ELSIF (F_BACnet_GetObjType(_ObjectId) <> BACnetObjectType_Group) THEN
	(* wrong mapping / invalid object ID *)
	IF _ObjectId = 0 THEN
		nErrorId := BACnet_ERR_WRONG_MAPPING;
	ELSE
		nErrorId := BACnet_ERR_INVALID_OBJECTID;
	END_IF
	bReady := FALSE;
	tObjectID := 16#FFFFFFFF;

ELSE
	(* clear error flag *)
	nErrorId := BACnet_ERR_NO_ERROR;
	(* ready state *)
	bReady := TRUE;
	tObjectID := _ObjectId;
END_IF

(* set error flag *)
bError := (nErrorId <> BACnet_ERR_NO_ERROR);

END_FUNCTION_BLOCK

// POUs/BACnet Objects/Remote (Client)/Extended Process Data/FB_BACnet_RemoteLoop_EX
FUNCTION_BLOCK FB_BACnet_RemoteLoop_EX
VAR_IN_OUT
	RemoteDevice		: FB_BACnet_RemoteDevice;
END_VAR
VAR_OUTPUT
	bReady				: BOOL;
	fControlledValue	: REAL;
	fPresentValue		: REAL;
	bOverridden			: BOOL;
	bOutOfService		: BOOL;
	bFault				: BOOL;
	bInAlarm			: BOOL;
	bOpenLoop			: BOOL;
	bOtherFault			: BOOL;
	eEventState			: E_BACNETEVENTSTATE;
	tObjectID			: T_BACnet_ObjectIdentifier := 16#FFFFFFFF;
	bError				: BOOL;
	nErrorId			: UINT;
END_VAR
VAR
	_PresentValue AT%I*: REAL; 			(* ~(BACnet_PresentValue 				: LP	: )
			                               	(BACnet_RemoteCycletimeRead 		: 1000	: )
											(BACnet_RemoteFlagsRead        		: 1     : )
                                   			(BACnet_RemoteResubscriptionInterval: 240 	: )
		                                	(BACnet_RemoteCycleTimeWrite   		: 1000	: )
		                                	(BACnet_RemoteFlagsWrite       		: 1		: )	*)
	_ControlledVariableValue AT%I*: REAL;(* ~(BACnet_ControlledVariableValue 	:		: )	*)
	_ObjectId AT%I*: DWORD;				(* ~(BACnet_ObjectIdentifier			:		: LINK) *)
	_Reliability AT%I*: WORD;; 			(* ~(BACnet_Reliability 				:		: )	*)
	_StatusFlags AT%I*: WORD; 			(* ~(BACnet_StatusFlags 				:		: )	*)
	_EventState AT%I*: WORD;			(* ~(BACnet_EventState					:		: )	*)
	_nUpdateCount : UDINT := 0;
	_StatusFlagsBits : ST_BACnet_StatusFlags;
END_VAR

(* update client device *)
IF RemoteDevice._nUpdateCount = _nUpdateCount THEN
	RemoteDevice();
END_IF
(* remind current number of update counter *)
_nUpdateCount := RemoteDevice._nUpdateCount;

IF NOT RemoteDevice.bOperational THEN
	nErrorId := BACnet_ERR_OPERATIONAL;
	bReady := FALSE;

ELSIF (F_BACnet_GetObjType(_ObjectId) <> BACnetObjectType_Loop) THEN
	(* wrong mapping / invalid object ID *)
	IF _ObjectId = 0 THEN
		nErrorId := BACnet_ERR_WRONG_MAPPING;
	ELSE
		nErrorId := BACnet_ERR_INVALID_OBJECTID;
	END_IF
	bReady := FALSE;
	tObjectID := 16#FFFFFFFF;

ELSIF _StatusFlags >= 4 THEN
	(* clear error flag *)
	nErrorId := BACnet_ERR_NO_ERROR;
	(* ready state *)
	bReady := TRUE;

	(* present value *)
	fPresentValue := _PresentValue;
	fControlledValue := _ControlledVariableValue;

	(* build bit states *)
	_StatusFlagsBits := F_BACnet_StatusFlags(_StatusFlags);

	(* copy states to output *)
	bOverridden := _StatusFlagsBits.overridden;
	bOutOfService := _StatusFlagsBits.out_of_service;
	bFault := _StatusFlagsBits.fault;
	bInAlarm := _StatusFlagsBits.in_alarm;
	bOpenLoop := (_Reliability = TO_WORD(BACnetReliability_open_loop));
	bOtherFault := (_Reliability = TO_WORD(BACnetReliability_unreliable_other));
	eEventState := TO_INT(_EventState);
	tObjectID := _ObjectId;
ELSE
	(* server device not ready, reset local ready also *)
	bReady := FALSE;
	(* and set error ID *)
	nErrorId := BACnet_ERR_WRONG_MAPPING;
END_IF

(* set error flag *)
bError := (nErrorId <> BACnet_ERR_NO_ERROR);

END_FUNCTION_BLOCK

// POUs/BACnet Objects/Remote (Client)/Extended Process Data/FB_BACnet_RemoteMultiStateInput_EX
FUNCTION_BLOCK FB_BACnet_RemoteMultiStateInput_EX
VAR_IN_OUT
	RemoteDevice		: FB_BACnet_RemoteDevice;
END_VAR
VAR_OUTPUT
	bReady				: BOOL;
	nPresentValue		: UDINT;
	bOverridden			: BOOL;
	bOutOfService		: BOOL;
	bFault				: BOOL;
	bInAlarm			: BOOL;
	bOverRange			: BOOL;
	bUnderRange			: BOOL;
	bNoSensor			: BOOL;
	bOpenLoop			: BOOL;
	bShortedLoop		: BOOL;
	bMultiStateFault	: BOOL;
	bOtherFault			: BOOL;
	eEventState			: E_BACNETEVENTSTATE;
	nNbrOfStates		: UDINT;
	tObjectID			: T_BACnet_ObjectIdentifier := 16#FFFFFFFF;
	bError				: BOOL;
	nErrorId			: UINT;
END_VAR
VAR
	_PresentValue AT%I*: UDINT; 		(* ~(BACnet_PresentValue 				:		: )
								   			(BACnet_ObjectType 					: MI	: )
											(BACnet_RemoteCycletimeRead 		: 1000	: )
											(BACnet_RemoteFlagsRead        		: 1		: )
											(BACnet_RemoteResubscriptionInterval: 240	: )
                                			(BACnet_RemoteCycleTimeWrite   		: 1000	: )
                                			(BACnet_RemoteFlagsWrite       		: 1		: )	*)
	_NumberOfStates AT%I*: UDINT;		(* ~(BACnet_NumberOfStates				:		: )	*)
	_ObjectId AT%I*: DWORD;				(* ~(BACnet_ObjectIdentifier			:		: LINK) *)
	_StatusFlags AT%I*: WORD; 			(* ~(BACnet_StatusFlags 				:		: )	*)
	_Reliability AT%I*: WORD;; 			(* ~(BACnet_Reliability 				:		: )	*)
	_EventState AT%I*: WORD; 			(* ~(BACnet_EventState 					:		: )	*)
	_nUpdateCount : UDINT := 0;
	_StatusFlagsBits : ST_BACnet_StatusFlags;
END_VAR

(* update client device *)
IF RemoteDevice._nUpdateCount = _nUpdateCount THEN
	RemoteDevice();
END_IF
(* remind current number of update counter *)
_nUpdateCount := RemoteDevice._nUpdateCount;

IF NOT RemoteDevice.bOperational THEN
	nErrorId := BACnet_ERR_OPERATIONAL;
	bReady := FALSE;

ELSIF (F_BACnet_GetObjType(_ObjectId) <> BACnetObjectType_MultiStateInput) THEN
	(* wrong mapping / invalid object ID *)
	IF _ObjectId = 0 THEN
		nErrorId := BACnet_ERR_WRONG_MAPPING;
	ELSE
		nErrorId := BACnet_ERR_INVALID_OBJECTID;
	END_IF
	bReady := FALSE;
	tObjectID := 16#FFFFFFFF;

ELSIF _StatusFlags >= 4 THEN
	(* clear error flag *)
	nErrorId := BACnet_ERR_NO_ERROR;
	(* ready state *)
	bReady := TRUE;

	(* present value *)
	nPresentValue := _PresentValue;

	(* build bit states *)
	_StatusFlagsBits := F_BACnet_StatusFlags(_StatusFlags);

	(* copy states to output *)
	bOverridden := _StatusFlagsBits.overridden;
	bOutOfService := _StatusFlagsBits.out_of_service;
	bFault := _StatusFlagsBits.fault;
	bInAlarm := _StatusFlagsBits.in_alarm;
	bOverRange := (_Reliability = TO_WORD(BACnetReliability_over_range));
	bUnderRange := (_Reliability = TO_WORD(BACnetReliability_under_range));
	bNoSensor := (_Reliability = TO_WORD(BACnetReliability_no_sensor));
	bOpenLoop := (_Reliability = TO_WORD(BACnetReliability_open_loop));
	bShortedLoop := (_Reliability = TO_WORD(BACnetReliability_shorted_loop));
	bMultiStateFault := (_Reliability = TO_WORD(BACnetReliability_multi_state_fault));
	bOtherFault := (_Reliability = TO_WORD(BACnetReliability_unreliable_other));
	nNbrOfStates := _NumberOfStates;
	eEventState := TO_INT(_EventState);
	tObjectID := _ObjectId;

ELSE
	(* server device not ready, reset local ready also *)
	bReady := FALSE;
	(* and set error ID *)
	nErrorId := BACnet_ERR_WRONG_MAPPING;
END_IF

(* set error flag *)
bError := (nErrorId <> BACnet_ERR_NO_ERROR);

END_FUNCTION_BLOCK

// POUs/BACnet Objects/Remote (Client)/Extended Process Data/FB_BACnet_RemoteMultiStateOutput_EX
FUNCTION_BLOCK FB_BACnet_RemoteMultiStateOutput_EX
VAR_INPUT
	bEnablePV			: BOOL; (* enable present value with priority x in priority array, FALSE = priority x disable *)
	bNullPV				: BOOL; (* clear priority entry *)
	nPV					: UDINT; (* number for priority x, when input bEnablePV is TRUE *)
END_VAR
VAR_IN_OUT
	RemoteDevice		: FB_BACnet_RemoteDevice;
END_VAR
VAR_OUTPUT
	bReady				: BOOL;
	nPresentValue		: UDINT;
	bOverridden			: BOOL;
	bOutOfService		: BOOL;
	bFault				: BOOL;
	bInAlarm			: BOOL;
	bNoOutput			: BOOL;
	bOpenLoop			: BOOL;
	bShortedLoop		: BOOL;
	bOtherFault			: BOOL;
	eEventState			: E_BACNETEVENTSTATE;
	nActivePrio			: UINT;
	nNbrOfStates		: UDINT;
	tObjectID			: T_BACnet_ObjectIdentifier := 16#FFFFFFFF;
	bError				: BOOL;
	nErrorId			: UINT;
END_VAR
VAR
	_PresentValue AT%I*: UDINT; 		(* ~(BACnet_PresentValue 				:		: )
								   			(BACnet_ObjectType					: MO	: )
											(BACnet_RemoteCycletimeRead 		: 1000	: )
											(BACnet_RemoteFlagsRead        		: 1		: )
											(BACnet_RemoteResubscriptionInterval: 240	: )
		                                	(BACnet_RemoteCycleTimeWrite   		: 1000	: )
		                                	(BACnet_RemoteFlagsWrite       		: 1		: )	*)
	_NumberOfStates AT%I*: UDINT;		(* ~(BACnet_NumberOfStates				:		: )	*)
	_ActivePriority AT%I*: UDINT; 		(* ~(BACnet_ActivePriority 				:		: )	*)
	_ObjectId AT%I*: DWORD;				(* ~(BACnet_ObjectIdentifier			:		: LINK) *)
	_StatusFlags AT%I*: WORD; 			(* ~(BACnet_StatusFlags					:		: )	*)
	_Reliability AT%I*: WORD;; 			(* ~(BACnet_Reliability					:		: )	*)
	_EventState AT%I*: WORD;			(* ~(BACnet_EventState					:		: )	*)
    _PresentValue_Priority12 AT%Q*: UDINT;(* ~(BACnet_PresentValue_Priority12	:		: )	*)
	_nUpdateCount : UDINT := 0;
	_StatusFlagsBits : ST_BACnet_StatusFlags;
END_VAR

(* update client device *)
IF RemoteDevice._nUpdateCount = _nUpdateCount THEN
	RemoteDevice();
END_IF
(* remind current number of update counter *)
_nUpdateCount := RemoteDevice._nUpdateCount;

IF RemoteDevice.bFirstCycle THEN
	(* first call of the server device since reboot/reset *)
	bReady := FALSE;
	_PresentValue_Priority12 := 16#FFFFFFFF;
ELSIF NOT RemoteDevice.bOperational THEN
	nErrorId := BACnet_ERR_OPERATIONAL;
	bReady := FALSE;

ELSIF (F_BACnet_GetObjType(_ObjectId) <> BACnetObjectType_MultiStateOutput) THEN
	(* wrong mapping / invalid object ID *)
	IF _ObjectId = 0 THEN
		nErrorId := BACnet_ERR_WRONG_MAPPING;
	ELSE
		nErrorId := BACnet_ERR_INVALID_OBJECTID;
	END_IF
	bReady := FALSE;
	tObjectID := 16#FFFFFFFF;

ELSIF _StatusFlags >= 4 THEN
	(* clear error flag *)
	nErrorId := BACnet_ERR_NO_ERROR;
	(* ready state *)
	bReady := TRUE;

	(* write into priority array *)
	_PresentValue_Priority12 := F_BACnet_MultiStatePV(bEnablePV, bNullPV, nPV);

	(* present value *)
	nPresentValue := _PresentValue;

	(* build bit states *)
	_StatusFlagsBits := F_BACnet_StatusFlags(_StatusFlags);

	(* copy states to output *)
	bOverridden := _StatusFlagsBits.overridden;
	bOutOfService := _StatusFlagsBits.out_of_service;
	bFault := _StatusFlagsBits.fault;
	bInAlarm := _StatusFlagsBits.in_alarm;
	bNoOutput := (_Reliability = TO_WORD(BACnetReliability_no_output));
	bOpenLoop := (_Reliability = TO_WORD(BACnetReliability_open_loop));
	bShortedLoop := (_Reliability = TO_WORD(BACnetReliability_shorted_loop));
	bOtherFault := (_Reliability = TO_WORD(BACnetReliability_unreliable_other));
	eEventState := TO_INT(_EventState);
	tObjectID := _ObjectId;

	(* copy active priority *)
	nActivePrio := UDINT_TO_UINT(_ActivePriority);

	(* number of states *)
	nNbrOfStates := _NumberOfStates;

ELSE
	(* server device not ready, reset local ready also *)
	bReady := FALSE;
	(* and set error ID *)
	nErrorId := BACnet_ERR_WRONG_MAPPING;
END_IF

(* set error flag *)
bError := (nErrorId <> BACnet_ERR_NO_ERROR);

END_FUNCTION_BLOCK

// POUs/BACnet Objects/Remote (Client)/Extended Process Data/FB_BACnet_RemoteMultiStateValue_EX
FUNCTION_BLOCK FB_BACnet_RemoteMultiStateValue_EX
VAR_INPUT
	bEnablePV			: BOOL; (* enable present value with priority x in priority array, FALSE = priority x disable *)
	bNullPV				: BOOL; (* clear priority entry *)
	nPV					: UDINT; (* number for priority x, when input bEnablePV is TRUE *)
END_VAR
VAR_IN_OUT
	RemoteDevice		: FB_BACnet_RemoteDevice;
END_VAR
VAR_OUTPUT
	bReady				: BOOL;
	nPresentValue		: UDINT;
	bOverridden			: BOOL;
	bOutOfService		: BOOL;
	bFault				: BOOL;
	bInAlarm			: BOOL;
	bMultiStateFault	: BOOL;
	bOtherFault			: BOOL;
	eEventState			: E_BACNETEVENTSTATE;
	nNbrOfStates		: UDINT;
	tObjectID			: T_BACnet_ObjectIdentifier := 16#FFFFFFFF;
	bError				: BOOL;
	nErrorId			: UINT;
END_VAR
VAR
	_PresentValue AT%I*: UDINT; 		(* ~(BACnet_PresentValue 				:		: )
											(BACnet_ObjectType 					: MV	: )
											(BACnet_RemoteCycletimeRead 		: 1000	: )
											(BACnet_RemoteFlagsRead        		: 1		: )
											(BACnet_RemoteResubscriptionInterval: 240	: )
											(BACnet_RemoteCycleTimeWrite   		: 1000	: )
											(BACnet_RemoteFlagsWrite       		: 1		: )	*)
	_NumberOfStates AT%I*: UDINT;		(* ~(BACnet_NumberOfStates				:		: )	*)
	_EventState AT%I*: WORD;			(* ~(BACnet_EventState					:		: )	*)
	_ObjectId AT%I*: DWORD;				(* ~(BACnet_ObjectIdentifier			:		: LINK) *)
	_StatusFlags AT%I*: WORD;			(* ~(BACnet_StatusFlags 				:		: )	*)
	_Reliability AT%I*: WORD;;			(* ~(BACnet_Reliability 				:		: )	*)
    _PresentValue_Priority12 AT%Q*: UDINT;(* ~(BACnet_PresentValue_Priority12	:		: )	*)
	_nUpdateCount : UDINT := 0;
	_StatusFlagsBits : ST_BACnet_StatusFlags;
END_VAR

(* update client device *)
IF RemoteDevice._nUpdateCount = _nUpdateCount THEN
	RemoteDevice();
END_IF
(* remind current number of update counter *)
_nUpdateCount := RemoteDevice._nUpdateCount;

IF RemoteDevice.bFirstCycle THEN
	(* first call of the server device since reboot/reset *)
	bReady := FALSE;
	_PresentValue_Priority12 := 16#FFFFFFFF;
ELSIF NOT RemoteDevice.bOperational THEN
	nErrorId := BACnet_ERR_OPERATIONAL;
	bReady := FALSE;

ELSIF (F_BACnet_GetObjType(_ObjectId) <> BACnetObjectType_MultiStateValue) THEN
	(* wrong mapping / invalid object ID *)
	IF _ObjectId = 0 THEN
		nErrorId := BACnet_ERR_WRONG_MAPPING;
	ELSE
		nErrorId := BACnet_ERR_INVALID_OBJECTID;
	END_IF
	bReady := FALSE;
	tObjectID := 16#FFFFFFFF;

ELSIF _StatusFlags >= 4 THEN
	(* clear error flag *)
	nErrorId := BACnet_ERR_NO_ERROR;
	(* ready state *)
	bReady := TRUE;

	(* write into priority array *)
	_PresentValue_Priority12 := F_BACnet_MultiStatePV(bEnablePV, bNullPV, nPV);

	(* present value *)
	nPresentValue := _PresentValue;

	(* build bit states *)
	_StatusFlagsBits := F_BACnet_StatusFlags(_StatusFlags);

	(* copy states to output *)
	bOverridden := _StatusFlagsBits.overridden;
	bOutOfService := _StatusFlagsBits.out_of_service;
	bFault := _StatusFlagsBits.fault;
	bInAlarm := _StatusFlagsBits.in_alarm;
	bMultiStateFault := (_Reliability = TO_WORD(BACnetReliability_multi_state_fault));
	bOtherFault := (_Reliability = TO_WORD(BACnetReliability_unreliable_other));
	eEventState := TO_INT(_EventState);
	tObjectID := _ObjectId;

	(* number of states *)
	nNbrOfStates := _NumberOfStates;

ELSE
	(* server device not ready, reset local ready also *)
	bReady := FALSE;
	(* and set error ID *)
	nErrorId := BACnet_ERR_WRONG_MAPPING;
END_IF

(* set error flag *)
bError := (nErrorId <> BACnet_ERR_NO_ERROR);

END_FUNCTION_BLOCK

// POUs/BACnet Objects/Remote (Client)/Extended Process Data/FB_BACnet_RemoteNotificationClass_EX
FUNCTION_BLOCK FB_BACnet_RemoteNotificationClass_EX
VAR_IN_OUT
	RemoteDevice		: FB_BACnet_RemoteDevice;
END_VAR
VAR_OUTPUT
	bReady				: BOOL;
	tObjectID			: T_BACnet_ObjectIdentifier := 16#FFFFFFFF;
	bError				: BOOL;
	nErrorId			: UINT;
END_VAR
VAR
	_ObjectId AT%I*: DWORD;				(* ~(BACnet_ObjectIdentifier	:		: LINK)
											(BACNET_OBJECTTYPE			: NC	: ) *)
	_nUpdateCount : UDINT := 0;
END_VAR

(* update client device *)
IF RemoteDevice._nUpdateCount = _nUpdateCount THEN
	RemoteDevice();
END_IF
(* remind current number of update counter *)
_nUpdateCount := RemoteDevice._nUpdateCount;

IF NOT RemoteDevice.bOperational THEN
	(* server device not ready, reset local ready also *)
	bReady := FALSE;
	(* and set error ID *)
	nErrorId := BACnet_ERR_OPERATIONAL;

ELSIF (F_BACnet_GetObjType(_ObjectId) <> BACnetObjectType_NotificationClass) THEN
	(* wrong mapping / invalid object ID *)
	IF _ObjectId = 0 THEN
		nErrorId := BACnet_ERR_WRONG_MAPPING;
	ELSE
		nErrorId := BACnet_ERR_INVALID_OBJECTID;
	END_IF
	bReady := FALSE;
	tObjectID := 16#FFFFFFFF;

ELSIF RemoteDevice.bOperational THEN
	(* clear error flag *)
	nErrorId := BACnet_ERR_NO_ERROR;
	(* ready state *)
	bReady := TRUE;
	tObjectID := _ObjectId;

END_IF

(* set error flag *)
bError := (nErrorId <> BACnet_ERR_NO_ERROR);

END_FUNCTION_BLOCK

// POUs/BACnet Objects/Remote (Client)/Extended Process Data/FB_BACnet_RemoteProgram_EX
FUNCTION_BLOCK FB_BACnet_RemoteProgram_EX
VAR_INPUT
	bEnablePV			: BOOL;
	ePV					: E_BACNETPROGRAMREQUEST;
	bRetrigger			: BOOL; (* execute selected request on raising edge again *)
END_VAR
VAR_IN_OUT
	RemoteDevice		: FB_BACnet_RemoteDevice;
END_VAR
VAR_OUTPUT
	bReady				: BOOL;
	ePrgState			: E_BACNETPROGRAMSTATE;
	ePrgChangeReq		: E_BACNETPROGRAMREQUEST;
	ePrgReasonHalt		: E_BACNETPROGRAMERROR;
	bOverridden			: BOOL;
	bOutOfService		: BOOL;
	bFault				: BOOL;
	bInAlarm			: BOOL;
	bProcessError		: BOOL;
	bOtherFault			: BOOL;
	tObjectID		: T_BACnet_ObjectIdentifier := 16#FFFFFFFF;
	bError				: BOOL;
	nErrorId			: UINT;
END_VAR
VAR
	_ProgramState AT%I*: WORD;			(* ~(BACnet_ProgramState 				:		: )
											(BACnet_ObjectType 					: PROG	: )
											(BACnet_RemoteCycletimeRead 		: 1000	: )
											(BACnet_RemoteFlagsRead        		: 1    	: )
											(BACnet_RemoteResubscriptionInterval: 240 	: )
											(BACnet_RemoteCycleTimeWrite   		: 1000	: )
											(BACnet_RemoteFlagsWrite       		: 1		: )	*)
	_ProgramChangeState AT%I*: WORD;	(* ~(BACnet_ProgramChange 				:		: )	*)
	_ReasonForHalt AT%I*: WORD;			(* ~(BACnet_ReasonForHalt 				: 		: )	*)
	_StatusFlags AT%I*: WORD;			(* ~(BACnet_StatusFlags 				:		: )	*)
	_Reliability AT%I*: WORD;;			(* ~(BACnet_Reliability 				:		: )	*)
	_ProgramChangeRequest AT%Q*: WORD;	(* ~(BACnet_ProgramChange 				:		: )	*)
	_ObjectId AT%I*: DWORD;				(* ~(BACnet_ObjectIdentifier			:		: LINK) *)
	_nUpdateCount : UDINT := 0;
	_StatusFlagsBits : ST_BACnet_StatusFlags;
	_rtrigRetriggerPv : R_TRIG;
END_VAR

(* update client device *)
IF RemoteDevice._nUpdateCount = _nUpdateCount THEN
	RemoteDevice();
END_IF
(* remind current number of update counter *)
_nUpdateCount := RemoteDevice._nUpdateCount;

(* call trigger *)
_rtrigRetriggerPv(CLK:= bRetrigger, Q=> );

IF RemoteDevice.bFirstCycle THEN
	(* first call of the server device since reboot/reset *)
	bReady := FALSE;
	_ProgramChangeRequest := 0;
ELSIF NOT RemoteDevice.bOperational THEN
	nErrorId := BACnet_ERR_OPERATIONAL;
	bReady := FALSE;

ELSIF (F_BACnet_GetObjType(_ObjectId) <> BACnetObjectType_Program) THEN
	(* wrong mapping / invalid object ID *)
	IF _ObjectId = 0 THEN
		nErrorId := BACnet_ERR_WRONG_MAPPING;
	ELSE
		nErrorId := BACnet_ERR_INVALID_OBJECTID;
	END_IF
	bReady := FALSE;
	tObjectID := 16#FFFFFFFF;

ELSIF _StatusFlags >= 4 THEN
	(* clear error flag *)
	nErrorId := BACnet_ERR_NO_ERROR;

	(* ready state *)
	bReady := TRUE;

	(* decode status flags *)
	_StatusFlagsBits := F_BACnet_StatusFlags(_StatusFlags);

	(* copy states to output *)
	bOverridden := _StatusFlagsBits.overridden;
	bOutOfService := _StatusFlagsBits.out_of_service;
	bFault := _StatusFlagsBits.fault;
	bInAlarm := _StatusFlagsBits.in_alarm;
	bProcessError := (_Reliability = TO_WORD(BACnetReliability_process_error));
	bOtherFault := (_Reliability = TO_WORD(BACnetReliability_unreliable_other));
	tObjectID := _ObjectId;

	(* present value from BACnet *)
	ePrgState := TO_INT(_ProgramState);
	(* present value to BACnet *)
	IF bEnablePV THEN
		IF _rtrigRetriggerPv.Q THEN
			(* trigger request *)
			_ProgramChangeRequest := 0;
		ELSE
			(* set request value *)
			_ProgramChangeRequest := TO_WORD(ePV);
		END_IF
	ELSE
		_ProgramChangeRequest := 0;
	END_IF
	(* other states *)
	ePrgReasonHalt := TO_INT(_ReasonForHalt);
	ePrgChangeReq := TO_INT(_ProgramChangeState);

ELSE
	(* server device not ready, reset local ready also *)
	bReady := FALSE;
	(* and set error ID *)
	nErrorId := BACnet_ERR_WRONG_MAPPING;
END_IF

(* set error flag *)
bError := (nErrorId <> BACnet_ERR_NO_ERROR);

END_FUNCTION_BLOCK

// POUs/BACnet Objects/Remote (Client)/Extended Process Data/FB_BACnet_RemotePulseConverter_EX
FUNCTION_BLOCK FB_BACnet_RemotePulseConverter_EX
VAR_IN_OUT
	RemoteDevice	: FB_BACnet_RemoteDevice;
END_VAR
VAR_OUTPUT
	bReady			: BOOL;
	fPresentValue	: REAL;
	nCount			: UDINT;
	bOverridden		: BOOL;
	bOutOfService	: BOOL;
	bFault			: BOOL;
	bInAlarm		: BOOL;
	bOverRange		: BOOL;
	bUnderRange		: BOOL;
	bNoSensor		: BOOL;
	bOpenLoop		: BOOL;
	bShortedLoop	: BOOL;
	bCommFailure	: BOOL;
	bConfigError	: BOOL;
	bOtherFault		: BOOL;
	tObjectID		: T_BACnet_ObjectIdentifier := 16#FFFFFFFF;
	bError			: BOOL;
	nErrorId		: UINT;
END_VAR
VAR
	_ObjectId AT%I*: DWORD;		(* ~(BACnet_ObjectIdentifier			:		: LINK) *)
	_Count AT%I*: UDINT;		(* ~(BACnet_Count		 				:		: ) *)
	_PresentValue AT%I*: REAL;	(* ~(BACnet_PresentValue 				:		: )	*)
	_StatusFlags AT%I*: UINT;	(* ~(BACnet_StatusFlags 				:		: )
									(BACnet_ObjectType 					: PC	: )
									(BACnet_RemoteCycletimeRead 		: 1000	: )
									(BACnet_RemoteFlagsRead        		: 1		: )
									(BACnet_RemoteResubscriptionInterval: 240	: )
                                	(BACnet_RemoteCycleTimeWrite   		: 1000	: )
                                	(BACnet_RemoteFlagsWrite       		: 1		: )	*)
	_Reliability AT%I*:WORD;	(* ~(BACnet_Reliability					:		: )	*)
	_StatusFlagsBits : ST_BACnet_StatusFlags;
	_nUpdateCount : UDINT := 0;
END_VAR

(* update client device *)
IF RemoteDevice._nUpdateCount = _nUpdateCount THEN
	RemoteDevice();
END_IF
(* remind current number of update counter *)
_nUpdateCount := RemoteDevice._nUpdateCount;

IF NOT RemoteDevice.bOperational THEN
	nErrorId := BACnet_ERR_OPERATIONAL;
	bReady := FALSE;

ELSIF (F_BACnet_GetObjType(_ObjectId) <> BACnetObjectType_PulseConverter) THEN
	(* wrong mapping / invalid object ID *)
	IF _ObjectId = 0 THEN
		nErrorId := BACnet_ERR_WRONG_MAPPING;
	ELSE
		nErrorId := BACnet_ERR_INVALID_OBJECTID;
	END_IF
	bReady := FALSE;
	tObjectID := 16#FFFFFFFF;

ELSIF _StatusFlags >= 4 THEN
	(* clear error flag *)
	nErrorId := BACnet_ERR_NO_ERROR;
	(* ready state *)
	bReady := TRUE;

	(* present value *)
	fPresentValue := _PresentValue;
	nCount := _Count;

	(* build bit states *)
	_StatusFlagsBits := F_BACnet_StatusFlags(_StatusFlags);

	(* copy states to output *)
	bOverridden := _StatusFlagsBits.overridden;
	bOutOfService := _StatusFlagsBits.out_of_service;
	bFault := _StatusFlagsBits.fault;
	bInAlarm := _StatusFlagsBits.in_alarm;
	tObjectID := _ObjectId;

	(* reliability *)
	bOverRange	:= (_Reliability = TO_WORD(BACnetReliability_over_range));
	bUnderRange	:= (_Reliability = TO_WORD(BACnetReliability_under_range));
	bNoSensor	:= (_Reliability = TO_WORD(BACnetReliability_no_sensor));
	bOpenLoop	:= (_Reliability = TO_WORD(BACnetReliability_open_loop));
	bShortedLoop:= (_Reliability = TO_WORD(BACnetReliability_shorted_loop));
	bCommFailure := (_Reliability = TO_WORD(BACnetReliability_communication_failure));
	bConfigError:= (_Reliability = TO_WORD(BACnetReliability_configuration_error));
	bOtherFault	:= (_Reliability = TO_WORD(BACnetReliability_unreliable_other));

ELSE
	(* server device not ready, reset local ready also *)
	bReady := FALSE;
	(* and set error ID *)
	nErrorId := BACnet_ERR_WRONG_MAPPING;
END_IF

(* set error flag *)
bError := (nErrorId <> BACnet_ERR_NO_ERROR);

END_FUNCTION_BLOCK

// POUs/BACnet Objects/Remote (Client)/Extended Process Data/FB_BACnet_RemoteSchedule_EX
FUNCTION_BLOCK FB_BACnet_RemoteSchedule_EX
VAR_IN_OUT
	RemoteDevice			: FB_BACnet_RemoteDevice;
END_VAR
VAR_OUTPUT
	bReady				: BOOL;
	bPresentValue		: BOOL;
	bOverridden			: BOOL;
	bOutOfService		: BOOL;
	bFault				: BOOL;
	bInAlarm			: BOOL;
	bConfigError		: BOOL;
	bOtherFault			: BOOL;
	tObjectID			: T_BACnet_ObjectIdentifier := 16#FFFFFFFF;
	bError				: BOOL;
	nErrorId			: UINT;
END_VAR
VAR
	_ObjectId AT%I*: DWORD;				(* ~(BACnet_ObjectIdentifier			:		: LINK) *)
	_Reliability AT%I*: WORD;; 			(* ~(BACnet_Reliability 				:		: )	*)
	_StatusFlags AT%I*: WORD; 			(* ~(BACnet_StatusFlags 				:		: )	*)
	_PresentValue AT%I*: BOOL;			(* ~(BACnet_PresentValueBool 			:		: )
											(BACnet_ObjectType 					: SCHED	: )
											(BACnet_RemoteCycletimeRead 		: 1000	: )
											(BACnet_RemoteFlagsRead        		: 1		: )
											(BACnet_RemoteResubscriptionInterval: 240	: )
                            				(BACnet_RemoteCycleTimeWrite   		: 1000	: )
                            				(BACnet_RemoteFlagsWrite       		: 1		: )	*)
	_StatusFlagsBits : ST_BACnet_StatusFlags;
	_nUpdateCount : UDINT := 0;
END_VAR

(* update client device *)
IF RemoteDevice._nUpdateCount = _nUpdateCount THEN
	RemoteDevice();
END_IF
(* remind current number of update counter *)
_nUpdateCount := RemoteDevice._nUpdateCount;

IF NOT RemoteDevice.bOperational THEN
	nErrorId := BACnet_ERR_OPERATIONAL;
	bReady := FALSE;

ELSIF (F_BACnet_GetObjType(_ObjectId) <> BACnetObjectType_Schedule) THEN
	(* wrong mapping / invalid object ID *)
	IF _ObjectId = 0 THEN
		nErrorId := BACnet_ERR_WRONG_MAPPING;
	ELSE
		nErrorId := BACnet_ERR_INVALID_OBJECTID;
	END_IF
	bReady := FALSE;
	tObjectID := 16#FFFFFFFF;

ELSIF _StatusFlags >= 4 THEN
	(* clear error flag *)
	nErrorId := BACnet_ERR_NO_ERROR;
	(* ready state *)
	bReady := TRUE;

	(* present value *)
	bPresentValue := _PresentValue;

	(* build bit states *)
	_StatusFlagsBits := F_BACnet_StatusFlags(_StatusFlags);

	(* copy states to output *)
	bOverridden := _StatusFlagsBits.overridden;
	bOutOfService := _StatusFlagsBits.out_of_service;
	bFault := _StatusFlagsBits.fault;
	bInAlarm := _StatusFlagsBits.in_alarm;
	bConfigError := (_Reliability = TO_WORD(BACnetReliability_configuration_error));
	bOtherFault := (_Reliability = TO_WORD(BACnetReliability_unreliable_other));
	tObjectID := _ObjectId;

ELSE
	bReady := FALSE;
	(* and set error ID *)
	nErrorId := BACnet_ERR_WRONG_MAPPING;
END_IF

(* set error flag *)
bError := (nErrorId <> BACnet_ERR_NO_ERROR);

END_FUNCTION_BLOCK

// POUs/BACnet Objects/Remote (Client)/Extended Process Data/FB_BACnet_RemoteTrendLog_EX
FUNCTION_BLOCK FB_BACnet_RemoteTrendLog_EX
VAR_OUTPUT
	bReady				: BOOL;
	bLogEnable			: BOOL;
	nRecordCount		: UDINT;
	nTotalCount			: UDINT;
	eEventState			: E_BACNETEVENTSTATE;
	tObjectID			: T_BACnet_ObjectIdentifier := 16#FFFFFFFF;
	bError				: BOOL;
	nErrorId			: UINT;
END_VAR
VAR_IN_OUT
	RemoteDevice			: FB_BACnet_RemoteDevice;
END_VAR
VAR
	_RecordCount AT%I*: UDINT;			(* ~(BACnet_RecordCount					:		: )
											(BACnet_ObjectType					: TLOG	: )
											(BACnet_RemoteCycletimeRead 		: 1000	: )
											(BACnet_RemoteFlagsRead        		: 1		: )
											(BACnet_RemoteResubscriptionInterval: 240	: )
											(BACnet_RemoteCycleTimeWrite   		: 1000	: )
                                			(BACnet_RemoteFlagsWrite       		: 1		: )	*)
	_TotalRecordCount AT%I*: UDINT;		(* ~(BACnet_TotalRecordCount			:		: )	*)
	_ObjectId AT%I*: DWORD;				(* ~(BACnet_ObjectIdentifier			:		: LINK) *)
	_EventState AT%I*: WORD;			(* ~(BACnet_EventState					:		: )	*)
	_LogEnable AT%I*: BOOL;				(* ~(BACnet_LogEnable					: 		: )	*)
	_nUpdateCount : UDINT := 0;
END_VAR

(* update client device *)
IF RemoteDevice._nUpdateCount = _nUpdateCount THEN
	RemoteDevice();
END_IF
(* remind current number of update counter *)
_nUpdateCount := RemoteDevice._nUpdateCount;

IF NOT RemoteDevice.bOperational THEN
	(* mapping seems to be wrong *)
	nErrorId := BACnet_ERR_OPERATIONAL;
	bReady := FALSE;

ELSIF (F_BACnet_GetObjType(_ObjectId) <> BACnetObjectType_TrendLog) THEN
	(* wrong mapping / invalid object ID *)
	IF _ObjectId = 0 THEN
		nErrorId := BACnet_ERR_WRONG_MAPPING;
	ELSE
		nErrorId := BACnet_ERR_INVALID_OBJECTID;
	END_IF
	bReady := FALSE;
	tObjectID := 16#FFFFFFFF;

ELSIF _EventState >= 0 THEN
	(* clear error flag *)
	nErrorId := BACnet_ERR_NO_ERROR;
	(* ready state *)
	bReady := TRUE;

	(* convert enumeration *)
	eEventState := TO_INT(_EventState);

	(* other states *)
	nRecordCount := _RecordCount;
	nTotalCount := _TotalRecordCount;
	bLogEnable := _LogEnable;
	tObjectID := _ObjectId;

ELSE
	bReady := FALSE;
	(* and set error ID *)
	nErrorId := BACnet_ERR_WRONG_MAPPING;
END_IF

(* set error flag *)
bError := (nErrorId <> BACnet_ERR_NO_ERROR);

END_FUNCTION_BLOCK

// POUs/BACnet Objects/Remote (Client)/WRITE/FB_BACnet_RemoteAnalogOutput_WR
FUNCTION_BLOCK FB_BACnet_RemoteAnalogOutput_WR
VAR_INPUT
	bEnablePV			: BOOL; (* enable present value with priority x in priority array, FALSE = priority x disable *)
	bNullPV				: BOOL; (* clear priority entry *)
	fPV					: REAL; (* decimal number for priority x, when input bEnablePV is TRUE *)
END_VAR
VAR_IN_OUT
	RemoteDevice		: FB_BACnet_RemoteDevice;
END_VAR
VAR_OUTPUT
	bReady				: BOOL;
	fPresentValue		: REAL;
	bOverridden			: BOOL;
	bOutOfService		: BOOL;
	bFault				: BOOL;
	bInAlarm			: BOOL;
	bError				: BOOL;
	nErrorId			: UINT;
END_VAR
VAR
	_PresentValue AT%I*: REAL; 			(* ~(BACnet_PresentValue 				:		: )
								   			(BACnet_ObjectType 					: AO	: )
											(BACnet_RemoteCycletimeRead 		: 1000	: )
											(BACnet_RemoteFlagsRead        		: 1		: )
											(BACnet_RemoteResubscriptionInterval: 240	: )
	                                		(BACnet_RemoteCycleTimeWrite   		: 1000	: )
	                                		(BACnet_RemoteFlagsWrite       		: 1		: )	*)
    _PresentValue_Priority12 AT%Q*: DWORD;(* ~(BACnet_PresentValue_Priority12	:		: )	*)
	_StatusFlags AT%I*: WORD; 			(* ~(BACnet_StatusFlags 				:		: )	*)
	_StatusFlagsBits : ST_BACnet_StatusFlags;

	_nUpdateCount : UDINT := 0;
END_VAR

(* update client device *)
IF RemoteDevice._nUpdateCount = _nUpdateCount THEN
	RemoteDevice();
END_IF
(* remind current number of update counter *)
_nUpdateCount := RemoteDevice._nUpdateCount;

IF RemoteDevice.bFirstCycle THEN
	(* first call of the server device since reboot/reset *)
	bReady := FALSE;
	_PresentValue_Priority12 := F_BACnet_RealNothing();
ELSIF NOT RemoteDevice.bOperational THEN
	nErrorId := BACnet_ERR_OPERATIONAL;
	bReady := FALSE;

ELSIF _StatusFlags >= 4 THEN
	(* clear error flag *)
	nErrorId := BACnet_ERR_NO_ERROR;
	(* ready state *)
	bReady := TRUE;

	(* write into priority array *)
	_PresentValue_Priority12 := F_BACnet_RealPV(bEnablePV, bNullPV, fPV);

	(* present value *)
	fPresentValue := _PresentValue;

	(* build bit states *)
	_StatusFlagsBits := F_BACnet_StatusFlags(_StatusFlags);

	(* copy states to output *)
	bOverridden := _StatusFlagsBits.overridden;
	bOutOfService := _StatusFlagsBits.out_of_service;
	bFault := _StatusFlagsBits.fault;
	bInAlarm := _StatusFlagsBits.in_alarm;
ELSE
	(* server device not ready, reset local ready also *)
	bReady := FALSE;
	(* and set error ID *)
	nErrorId := BACnet_ERR_WRONG_MAPPING;
END_IF

(* set error flag *)
bError := (nErrorId <> BACnet_ERR_NO_ERROR);

END_FUNCTION_BLOCK

// POUs/BACnet Objects/Remote (Client)/WRITE/FB_BACnet_RemoteAnalogValue_WR
FUNCTION_BLOCK FB_BACnet_RemoteAnalogValue_WR
VAR_INPUT
	bEnablePV			: BOOL; (* enable present value with priority x in priority array, FALSE = priority x disable *)
	bNullPV				: BOOL; (* clear priority entry *)
	fPV					: REAL; (* decimal number for priority x, when input bEnablePV is TRUE *)
END_VAR
VAR_IN_OUT
	RemoteDevice		: FB_BACnet_RemoteDevice;
END_VAR
VAR_OUTPUT
	bReady				: BOOL;
	fPresentValue		: REAL;
	bOverridden			: BOOL;
	bOutOfService		: BOOL;
	bFault				: BOOL;
	bInAlarm			: BOOL;
	bError				: BOOL;
	nErrorId			: UINT;
END_VAR
VAR
	_PresentValue AT%I*: REAL; 			(* ~(BACnet_PresentValue 				:		: )
								   			(BACnet_ObjectType 					: AV	: )
											(BACnet_RemoteCycletimeRead 		: 1000	: )
											(BACnet_RemoteFlagsRead        		: 1		: )
											(BACnet_RemoteResubscriptionInterval: 240	: )
	                                		(BACnet_RemoteCycleTimeWrite   		: 1000	: )
	                                		(BACnet_RemoteFlagsWrite       		: 1		: )	*)
    _PresentValue_Priority12 AT%Q*: DWORD;(* ~(BACnet_PresentValue_Priority12	:		: )	*)
	_StatusFlags AT%I*: WORD; 			(* ~(BACnet_StatusFlags 				:		: )	*)
	_StatusFlagsBits : ST_BACnet_StatusFlags;

	_nUpdateCount : UDINT := 0;
END_VAR

(* update client device *)
IF RemoteDevice._nUpdateCount = _nUpdateCount THEN
	RemoteDevice();
END_IF
(* remind current number of update counter *)
_nUpdateCount := RemoteDevice._nUpdateCount;

IF RemoteDevice.bFirstCycle THEN
	(* first call of the server device since reboot/reset *)
	bReady := FALSE;
	_PresentValue_Priority12 := F_BACnet_RealNothing();
ELSIF NOT RemoteDevice.bOperational THEN
	nErrorId := BACnet_ERR_OPERATIONAL;
	bReady := FALSE;

ELSIF _StatusFlags >= 4 THEN
	(* clear error flag *)
	nErrorId := BACnet_ERR_NO_ERROR;
	(* ready state *)
	bReady := TRUE;

	(* write into priority array *)
	_PresentValue_Priority12 := F_BACnet_RealPV(bEnablePV, bNullPV, fPV);

	(* present value *)
	fPresentValue := _PresentValue;

	(* build bit states *)
	_StatusFlagsBits := F_BACnet_StatusFlags(_StatusFlags);

	(* copy states to output *)
	bOverridden := _StatusFlagsBits.overridden;
	bOutOfService := _StatusFlagsBits.out_of_service;
	bFault := _StatusFlagsBits.fault;
	bInAlarm := _StatusFlagsBits.in_alarm;
ELSE
	(* server device not ready, reset local ready also *)
	bReady := FALSE;
	(* and set error ID *)
	nErrorId := BACnet_ERR_WRONG_MAPPING;
END_IF

(* set error flag *)
bError := (nErrorId <> BACnet_ERR_NO_ERROR);

END_FUNCTION_BLOCK

// POUs/BACnet Objects/Remote (Client)/WRITE/FB_BACnet_RemoteBinaryOutput_WR
FUNCTION_BLOCK FB_BACnet_RemoteBinaryOutput_WR
VAR_INPUT
	bEnablePV			: BOOL; (* enable present value with priority x in priority array, FALSE = priority x disable *)
	bNullPV				: BOOL; (* clear priority entry *)
	bPV					: BOOL; (* present value bool type *)
END_VAR
VAR_IN_OUT
	RemoteDevice		: FB_BACnet_RemoteDevice;
END_VAR
VAR_OUTPUT
	bReady				: BOOL;
	bPresentValue		: BOOL;
	bOverridden			: BOOL;
	bOutOfService		: BOOL;
	bFault				: BOOL;
	bInAlarm			: BOOL;
	bError				: BOOL;
	nErrorId			: UINT;
END_VAR
VAR
	_PresentValue AT%I*: WORD; 			(* ~(BACnet_PresentValue 				:		: )
								   			(BACnet_ObjectType 					: BO	: )
											(BACnet_RemoteCycletimeRead 		: 1000	: )
											(BACnet_RemoteFlagsRead        		: 1		: )
											(BACnet_RemoteResubscriptionInterval: 240	: )
		                            		(BACnet_RemoteCycleTimeWrite   		: 1000	: )
		                            		(BACnet_RemoteFlagsWrite       		: 1		: )	*)
    _PresentValue_Priority12 AT%Q*: WORD;(* ~(BACnet_PresentValue_Priority12	:		: )	*)
	_StatusFlags AT%I*: WORD; 			(* ~(BACnet_StatusFlags 				:		: )	*)
	_StatusFlagsBits : ST_BACnet_StatusFlags;
	_nUpdateCount : UDINT := 0;
END_VAR

(* update client device *)
IF RemoteDevice._nUpdateCount = _nUpdateCount THEN
	RemoteDevice();
END_IF
(* remind current number of update counter *)
_nUpdateCount := RemoteDevice._nUpdateCount;

IF RemoteDevice.bFirstCycle THEN
	(* first call of the server device since reboot/reset *)
	bReady := FALSE;
	_PresentValue_Priority12 := to_word(BACnetBinaryPV_Nothing);
ELSIF NOT RemoteDevice.bOperational THEN
	nErrorId := BACnet_ERR_OPERATIONAL;
	bReady := FALSE;

ELSIF _StatusFlags >= 4 THEN
	(* clear error flag *)
	nErrorId := BACnet_ERR_NO_ERROR;
	(* ready state *)
	bReady := TRUE;

	(* write into priority array *)
	_PresentValue_Priority12 := to_word(F_Bool_To_BinPV(bEnablePV, bNullPV, bPV));

	(* present value *)
	bPresentValue := F_BinPV_To_Bool(TO_INT(_PresentValue));

	(* build bit states *)
	_StatusFlagsBits := F_BACnet_StatusFlags(_StatusFlags);

	(* copy states to output *)
	bOverridden := _StatusFlagsBits.overridden;
	bOutOfService := _StatusFlagsBits.out_of_service;
	bFault := _StatusFlagsBits.fault;
	bInAlarm := _StatusFlagsBits.in_alarm;
ELSE
	(* server device not ready, reset local ready also *)
	bReady := FALSE;
	(* and set error ID *)
	nErrorId := BACnet_ERR_WRONG_MAPPING;
END_IF

(* set error flag *)
bError := (nErrorId <> BACnet_ERR_NO_ERROR);

END_FUNCTION_BLOCK

// POUs/BACnet Objects/Remote (Client)/WRITE/FB_BACnet_RemoteBinaryValue_WR
FUNCTION_BLOCK FB_BACnet_RemoteBinaryValue_WR
VAR_INPUT
	bEnablePV			: BOOL; (* enable present value with priority x in priority array, FALSE = priority x disable *)
	bNullPV				: BOOL; (* clear priority entry *)
	bPV					: BOOL; (* present value bool type *)
END_VAR
VAR_IN_OUT
	RemoteDevice		: FB_BACnet_RemoteDevice;
END_VAR
VAR_OUTPUT
	bReady				: BOOL;
	bPresentValue		: BOOL;
	bOverridden			: BOOL;
	bOutOfService		: BOOL;
	bFault				: BOOL;
	bInAlarm			: BOOL;
	bError				: BOOL;
	nErrorId			: UINT;
END_VAR
VAR

	_PresentValue AT%I*: WORD; 			(* ~(BACnet_PresentValue 				:		: )
								   			(BACnet_ObjectType 					: BV	: )
											(BACnet_RemoteCycletimeRead 		: 1000	: )
											(BACnet_RemoteFlagsRead        		: 1		: )
											(BACnet_RemoteResubscriptionInterval: 240	: )
	                                		(BACnet_RemoteCycleTimeWrite   		: 1000	: )
	                                		(BACnet_RemoteFlagsWrite       		: 1		: )	*)
    _PresentValue_Priority12 AT%Q*: WORD;(* ~(BACnet_PresentValue_Priority12	:		: )	*)
	_StatusFlags AT%I*: WORD; 			(* ~(BACnet_StatusFlags 				:		: )	*)
	_StatusFlagsBits : ST_BACnet_StatusFlags;

	_nUpdateCount : UDINT := 0;
END_VAR

(* update client device *)
IF RemoteDevice._nUpdateCount = _nUpdateCount THEN
	RemoteDevice();
END_IF
(* remind current number of update counter *)
_nUpdateCount := RemoteDevice._nUpdateCount;

IF RemoteDevice.bFirstCycle THEN
	(* first call of the server device since reboot/reset *)
	bReady := FALSE;
	_PresentValue_Priority12 := TO_WORD(BACnetBinaryPV_Nothing);
ELSIF NOT RemoteDevice.bOperational THEN
	nErrorId := BACnet_ERR_OPERATIONAL;
	bReady := FALSE;

ELSIF _StatusFlags >= 4 THEN
	(* clear error flag *)
	nErrorId := BACnet_ERR_NO_ERROR;
	(* ready state *)
	bReady := TRUE;

	(* write into priority array *)
	_PresentValue_Priority12 := to_word(F_Bool_To_BinPV(bEnablePV, bNullPV, bPV));

	(* present value *)
	bPresentValue := F_BinPV_To_Bool(TO_INT(_PresentValue));

	(* build bit states *)
	_StatusFlagsBits := F_BACnet_StatusFlags(_StatusFlags);

	(* copy states to output *)
	bOverridden := _StatusFlagsBits.overridden;
	bOutOfService := _StatusFlagsBits.out_of_service;
	bFault := _StatusFlagsBits.fault;
	bInAlarm := _StatusFlagsBits.in_alarm;

ELSE
	(* server device not ready, reset local ready also *)
	bReady := FALSE;
	(* and set error ID *)
	nErrorId := BACnet_ERR_WRONG_MAPPING;
END_IF

(* set error flag *)
bError := (nErrorId <> BACnet_ERR_NO_ERROR);

END_FUNCTION_BLOCK

// POUs/BACnet Objects/Remote (Client)/WRITE/FB_BACnet_RemoteCommand_WR
FUNCTION_BLOCK FB_BACnet_RemoteCommand_WR
VAR_INPUT
	bEnablePV			: BOOL;
	nPV					: UDINT;
	bRetrigger			: BOOL; (* execute selected action on raising edge again *)
END_VAR
VAR_IN_OUT
	RemoteDevice		: FB_BACnet_RemoteDevice;
END_VAR
VAR_OUTPUT
	bReady				: BOOL;
	nPresentValue		: UDINT;
	bAllWritesOk		: BOOL; (* all actions in selected action list are written *)
	bInProcess			: BOOL; (* object is busy *)
	bError				: BOOL;
	nErrorId			: UINT;
END_VAR
VAR
	_PresentValueIn AT%I*: UDINT; 		(* ~(BACnet_PresentValue 				:		: )
								   			(BACnet_ObjectType 					: CMD	: )
											(BACnet_RemoteCycletimeRead 		: 1000	: )
											(BACnet_RemoteFlagsRead        		: 1		: )
											(BACnet_RemoteResubscriptionInterval: 240	: )
	                                		(BACnet_RemoteCycleTimeWrite   		: 1000	: )
	                                		(BACnet_RemoteFlagsWrite       		: 1		: )	*)
	_InProcess AT%I*: BOOL;				(* ~(BACnet_InProcess 					:		: )	*)
	_AllWritesSuccessful AT%I*: BOOL;	(* ~(BACnet_AllWritesSuccessful			:		: )	*)
    _PresentValueOut AT%Q*: UDINT;		(* ~(BACnet_PresentValue	 	   		:      	: )	*)
	_nUpdateCount : UDINT := 0;
	_rtrigRetriggerPv : R_TRIG;
END_VAR

(* update client device *)
IF RemoteDevice._nUpdateCount = _nUpdateCount THEN
	RemoteDevice();
END_IF
(* remind current number of update counter *)
_nUpdateCount := RemoteDevice._nUpdateCount;

(* call trigger *)
_rtrigRetriggerPv(CLK:= bRetrigger, Q=> );

IF RemoteDevice.bOperational THEN
	(* clear error flag *)
	nErrorId := BACnet_ERR_NO_ERROR;
	(* ready state *)
	bReady := TRUE;
	(* present value from BACnet *)
	nPresentValue := _PresentValueIn;
	(* present value to BACnet *)
	IF bEnablePV THEN
		IF _rtrigRetriggerPv.Q THEN
			(* trigger action list *)
			_PresentValueOut := 0;
		ELSE
			(* set present value *)
			_PresentValueOut := nPV;
		END_IF
	ELSE
		(* deactivate mapped present value --> other objects can write to property *)
		_PresentValueOut := 16#0;
	END_IF
	(* other states *)
	bAllWritesOk := _AllWritesSuccessful;
	bInProcess := _InProcess;
ELSIF RemoteDevice.bFirstCycle THEN
	(* first call of the server device since reboot/reset *)
	bReady := FALSE;
	_PresentValueOut := 0;
ELSE
	(* server device not ready, reset local ready also *)
	bReady := FALSE;
	(* and set error ID *)
	nErrorId := BACnet_ERR_WRONG_MAPPING;
END_IF

(* set error flag *)
bError := (nErrorId <> BACnet_ERR_NO_ERROR);

END_FUNCTION_BLOCK

// POUs/BACnet Objects/Remote (Client)/WRITE/FB_BACnet_RemoteMultiStateOutput_WR
FUNCTION_BLOCK FB_BACnet_RemoteMultiStateOutput_WR
VAR_INPUT
	bEnablePV			: BOOL; (* enable present value with priority x in priority array, FALSE = priority x disable *)
	bNullPV				: BOOL; (* clear priority entry *)
	nPV					: UDINT; (* number for priority x, when input bEnablePV is TRUE *)
END_VAR
VAR_IN_OUT
	RemoteDevice		: FB_BACnet_RemoteDevice;
END_VAR
VAR_OUTPUT
	bReady				: BOOL;
	nPresentValue		: UDINT;
	bOverridden			: BOOL;
	bOutOfService		: BOOL;
	bFault				: BOOL;
	bInAlarm			: BOOL;
	nNbrOfStates		: UDINT;
	bError				: BOOL;
	nErrorId			: UINT;
END_VAR
VAR
	_PresentValue AT%I*: UDINT; 			(* ~(BACnet_PresentValue 				:		: )
								   				(BACnet_ObjectType					: MO	: )
												(BACnet_RemoteCycletimeRead 		: 1000	: )
												(BACnet_RemoteFlagsRead        		: 1		: )
												(BACnet_RemoteResubscriptionInterval: 240	: )
		                                		(BACnet_RemoteCycleTimeWrite   		: 1000	: )
		                                		(BACnet_RemoteFlagsWrite       		: 1		: )	*)
	_NumberOfStates AT%I*: UDINT;			(* ~(BACnet_NumberOfStates				:		: )	*)
	_StatusFlags AT%I*: WORD; 				(* ~(BACnet_StatusFlags					:		: )	*)
    _PresentValue_Priority12 AT%Q*: UDINT;	(* ~(BACnet_PresentValue_Priority12		:		: )	*)
	_StatusFlagsBits : ST_BACnet_StatusFlags;
	_nUpdateCount : UDINT := 0;
END_VAR

(* update client device *)
IF RemoteDevice._nUpdateCount = _nUpdateCount THEN
	RemoteDevice();
END_IF
(* remind current number of update counter *)
_nUpdateCount := RemoteDevice._nUpdateCount;

IF RemoteDevice.bFirstCycle THEN
	(* first call of the server device since reboot/reset *)
	bReady := FALSE;
	_PresentValue_Priority12 := 16#FFFFFFFF;
ELSIF NOT RemoteDevice.bOperational THEN
	nErrorId := BACnet_ERR_OPERATIONAL;
	bReady := FALSE;

ELSIF _StatusFlags >= 4 THEN
	(* clear error flag *)
	nErrorId := BACnet_ERR_NO_ERROR;
	(* ready state *)
	bReady := TRUE;

	(* write into priority array *)
	_PresentValue_Priority12 := F_BACnet_MultiStatePV(bEnablePV, bNullPV, nPV);

	(* present value *)
	nPresentValue := _PresentValue;

	(* build bit states *)
	_StatusFlagsBits := F_BACnet_StatusFlags(_StatusFlags);

	(* copy states to output *)
	bOverridden := _StatusFlagsBits.overridden;
	bOutOfService := _StatusFlagsBits.out_of_service;
	bFault := _StatusFlagsBits.fault;
	bInAlarm := _StatusFlagsBits.in_alarm;

	(* number of states *)
	nNbrOfStates := _NumberOfStates;

ELSE
	(* server device not ready, reset local ready also *)
	bReady := FALSE;
	(* and set error ID *)
	nErrorId := BACnet_ERR_WRONG_MAPPING;
END_IF

(* set error flag *)
bError := (nErrorId <> BACnet_ERR_NO_ERROR);

END_FUNCTION_BLOCK

// POUs/BACnet Objects/Remote (Client)/WRITE/FB_BACnet_RemoteMultiStateValue_WR
FUNCTION_BLOCK FB_BACnet_RemoteMultiStateValue_WR
VAR_INPUT
	bEnablePV			: BOOL; (* enable present value with priority x in priority array, FALSE = priority x disable *)
	bNullPV				: BOOL; (* clear priority entry *)
	nPV					: UDINT; (* number for priority x, when input bEnablePV is TRUE *)
END_VAR
VAR_IN_OUT
	RemoteDevice		: FB_BACnet_RemoteDevice;
END_VAR
VAR_OUTPUT
	bReady				: BOOL;
	nPresentValue		: UDINT;
	bOverridden			: BOOL;
	bOutOfService		: BOOL;
	bFault				: BOOL;
	bInAlarm			: BOOL;
	nNbrOfStates		: UDINT;
	bError				: BOOL;
	nErrorId			: UINT;
END_VAR
VAR
	_PresentValue AT%I*: UDINT; 			(* ~(BACnet_PresentValue 				:		: )
								   				(BACnet_ObjectType 					: MV	: )
												(BACnet_RemoteCycletimeRead 		: 1000	: )
												(BACnet_RemoteFlagsRead        		: 1		: )
												(BACnet_RemoteResubscriptionInterval: 240	: )
		                                		(BACnet_RemoteCycleTimeWrite   		: 1000	: )
		                                		(BACnet_RemoteFlagsWrite       		: 1		: )	*)
	_NumberOfStates AT%I*: UDINT;			(* ~(BACnet_NumberOfStates				:		: )	*)
	_StatusFlags AT%I*: WORD; 				(* ~(BACnet_StatusFlags 				:		: )	*)
    _PresentValue_Priority12 AT%Q*: UDINT;	(* ~(BACnet_PresentValue_Priority12		:		: )	*)
	_StatusFlagsBits : ST_BACnet_StatusFlags;
	_nUpdateCount : UDINT := 0;
END_VAR

(* update client device *)
IF RemoteDevice._nUpdateCount = _nUpdateCount THEN
	RemoteDevice();
END_IF
(* remind current number of update counter *)
_nUpdateCount := RemoteDevice._nUpdateCount;

IF RemoteDevice.bFirstCycle THEN
	(* first call of the server device since reboot/reset *)
	bReady := FALSE;
	_PresentValue_Priority12 := 16#FFFFFFFF;
ELSIF NOT RemoteDevice.bOperational THEN
	nErrorId := BACnet_ERR_OPERATIONAL;
	bReady := FALSE;

ELSIF _StatusFlags >= 4 THEN
	(* clear error flag *)
	nErrorId := BACnet_ERR_NO_ERROR;
	(* ready state *)
	bReady := TRUE;

	(* write into priority array *)
	_PresentValue_Priority12 := F_BACnet_MultiStatePV(bEnablePV, bNullPV, nPV);

	(* present value *)
	nPresentValue := _PresentValue;

	(* build bit states *)
	_StatusFlagsBits := F_BACnet_StatusFlags(_StatusFlags);

	(* copy states to output *)
	bOverridden := _StatusFlagsBits.overridden;
	bOutOfService := _StatusFlagsBits.out_of_service;
	bFault := _StatusFlagsBits.fault;
	bInAlarm := _StatusFlagsBits.in_alarm;

	(* number of states *)
	nNbrOfStates := _NumberOfStates;

ELSE
	(* server device not ready, reset local ready also *)
	bReady := FALSE;
	(* and set error ID *)
	nErrorId := BACnet_ERR_WRONG_MAPPING;
END_IF

(* set error flag *)
bError := (nErrorId <> BACnet_ERR_NO_ERROR);

END_FUNCTION_BLOCK

// POUs/BACnet Objects/Remote (Client)/WRITE/FB_BACnet_RemoteProgram_WR
FUNCTION_BLOCK FB_BACnet_RemoteProgram_WR
VAR_INPUT
	bEnablePV			: BOOL;
	ePV					: E_BACNETPROGRAMREQUEST;
	bRetrigger			: BOOL; (* execute selected request on raising edge again *)
END_VAR
VAR_IN_OUT
	RemoteDevice		: FB_BACnet_RemoteDevice;
END_VAR
VAR_OUTPUT
	bReady				: BOOL;
	ePrgState			: E_BACNETPROGRAMSTATE;
	ePrgReasonHalt		: E_BACNETPROGRAMERROR;
	bOverridden			: BOOL;
	bOutOfService		: BOOL;
	bFault				: BOOL;
	bInAlarm			: BOOL;
	bError				: BOOL;
	nErrorId			: UINT;
END_VAR
VAR
	_ProgramState AT%I*: WORD;			(* ~(BACnet_ProgramState 				:		: )
								   			(BACnet_ObjectType 					: PROG	: )
			                            	(BACnet_RemoteCycletimeRead 		: 1000	: )
											(BACnet_RemoteFlagsRead        		: 1    	: )
                                   			(BACnet_RemoteResubscriptionInterval: 240 	: )
	                                		(BACnet_RemoteCycleTimeWrite   		: 1000	: )
	                                		(BACnet_RemoteFlagsWrite       		: 1		: )	*)
	_ReasonForHalt AT%I*: WORD;			(* ~(BACnet_ReasonForHalt 				: 		: )	*)
	_StatusFlags AT%I*: WORD;			(* ~(BACnet_StatusFlags 				:		: )	*)
	_ProgramChangeRequest AT%Q*: WORD;	(* ~(BACnet_ProgramChange 				:		: )	*)
	_nUpdateCount : UDINT := 0;
	_StatusFlagsBits : ST_BACnet_StatusFlags;
	_rtrigRetriggerPv : R_TRIG;
END_VAR

(* update client device *)
IF RemoteDevice._nUpdateCount = _nUpdateCount THEN
	RemoteDevice();
END_IF
(* remind current number of update counter *)
_nUpdateCount := RemoteDevice._nUpdateCount;

(* call trigger *)
_rtrigRetriggerPv(CLK:= bRetrigger, Q=> );

IF RemoteDevice.bFirstCycle THEN
	(* first call of the server device since reboot/reset *)
	bReady := FALSE;
	_ProgramChangeRequest := 0;
ELSIF NOT RemoteDevice.bOperational THEN
	nErrorId := BACnet_ERR_OPERATIONAL;
	bReady := FALSE;

ELSIF _StatusFlags >= 4 THEN
	(* clear error flag *)
	nErrorId := BACnet_ERR_NO_ERROR;

	(* ready state *)
	bReady := TRUE;

	(* decode status flags *)
	_StatusFlagsBits := F_BACnet_StatusFlags(_StatusFlags);

	(* copy states to output *)
	bOverridden := _StatusFlagsBits.overridden;
	bOutOfService := _StatusFlagsBits.out_of_service;
	bFault := _StatusFlagsBits.fault;
	bInAlarm := _StatusFlagsBits.in_alarm;

	(* present value from BACnet *)
	ePrgState := TO_INT(_ProgramState);
	(* present value to BACnet *)
	IF bEnablePV THEN
		IF _rtrigRetriggerPv.Q THEN
			(* trigger request *)
			_ProgramChangeRequest := 0;
		ELSE
			(* set request value *)
			_ProgramChangeRequest := TO_WORD(ePV);
		END_IF
	ELSE
		_ProgramChangeRequest := 0;
	END_IF
	(* other states *)
	ePrgReasonHalt := to_int(_ReasonForHalt);
ELSE
	(* server device not ready, reset local ready also *)
	bReady := FALSE;
	(* and set error ID *)
	nErrorId := BACnet_ERR_WRONG_MAPPING;
END_IF

(* set error flag *)
bError := (nErrorId <> BACnet_ERR_NO_ERROR);

END_FUNCTION_BLOCK

// POUs/BACnet Objects/Remote (Client)/FB_BACnet_RemoteAccumulator
FUNCTION_BLOCK FB_BACnet_RemoteAccumulator
VAR_IN_OUT
	RemoteDevice		: FB_BACnet_RemoteDevice;
END_VAR
VAR_OUTPUT
	bReady				: BOOL;
	nPresentValue		: UDINT;
	bOverridden			: BOOL;
	bOutOfService		: BOOL;
	bFault				: BOOL;
	bInAlarm			: BOOL;
	bError				: BOOL;
	nErrorId			: UINT;
END_VAR
VAR
	_PresentValue AT%I*:UDINT;		(* ~(BACnet_PresentValue				:		: )
										(BACnet_ObjectType					: ACC	: )
										(BACnet_RemoteCycletimeRead			: 1000	: )
										(BACnet_RemoteFlagsRead				: 1		: )
										(BACnet_RemoteResubscriptionInterval: 240	: )
                                		(BACnet_RemoteCycleTimeWrite   		: 1000	: )
                                		(BACnet_RemoteFlagsWrite       		: 1		: )	*)
	_StatusFlags AT%I*:WORD;		(* ~(BACnet_StatusFlags					:		: )	*)
	_StatusFlagsBits : ST_BACnet_StatusFlags;

	_nUpdateCount : UDINT := 0;
END_VAR

(* update client device *)
IF RemoteDevice._nUpdateCount = _nUpdateCount THEN
	RemoteDevice();
END_IF
(* remind current number of update counter *)
_nUpdateCount := RemoteDevice._nUpdateCount;

IF NOT RemoteDevice.bOperational THEN
	nErrorId := BACnet_ERR_OPERATIONAL;
	bReady := FALSE;

ELSIF _StatusFlags >= 4 THEN
	(* clear error flag *)
	nErrorId := BACnet_ERR_NO_ERROR;
	bReady := TRUE;
	(* copy present value *)
	nPresentValue := _PresentValue;

	(* build bit states *)
	_StatusFlagsBits := F_BACnet_StatusFlags(_StatusFlags);

	(* copy states to output *)
	bOverridden := _StatusFlagsBits.overridden;
	bOutOfService := _StatusFlagsBits.out_of_service;
	bFault := _StatusFlagsBits.fault;
	bInAlarm := _StatusFlagsBits.in_alarm;
ELSE
	bReady := FALSE;
	(* and set error ID *)
	nErrorId := BACnet_ERR_WRONG_MAPPING;
END_IF

(* set error flag *)
bError := (nErrorId <> BACnet_ERR_NO_ERROR);

END_FUNCTION_BLOCK

// POUs/BACnet Objects/Remote (Client)/FB_BACnet_RemoteAnalogInput
FUNCTION_BLOCK FB_BACnet_RemoteAnalogInput
VAR_IN_OUT
	RemoteDevice			: FB_BACnet_RemoteDevice;
END_VAR
VAR_OUTPUT
	bReady				: BOOL;
	fPresentValue		: REAL;
	bOverridden			: BOOL;
	bOutOfService		: BOOL;
	bFault				: BOOL;
	bInAlarm			: BOOL;
	bError				: BOOL;
	nErrorId			: UINT;
END_VAR
VAR
	_PresentValue AT%I*: REAL; 			(* ~(BACnet_PresentValue 				:		: )
								   			(BACnet_ObjectType 					: AI	: )
											(BACnet_RemoteCycletimeRead 		: 1000	: )
											(BACnet_RemoteFlagsRead        		: 1		: )
											(BACnet_RemoteResubscriptionInterval: 240	: )
	                                		(BACnet_RemoteCycleTimeWrite   		: 1000	: )
	                                		(BACnet_RemoteFlagsWrite       		: 1		: )	*)
	_StatusFlags AT%I*: WORD; 			(* ~(BACnet_StatusFlags 				:		: )	*)
	_StatusFlagsBits : ST_BACnet_StatusFlags;

	_nUpdateCount : UDINT := 0;
END_VAR

(* update client device *)
IF RemoteDevice._nUpdateCount = _nUpdateCount THEN
	RemoteDevice();
END_IF
(* remind current number of update counter *)
_nUpdateCount := RemoteDevice._nUpdateCount;

IF NOT RemoteDevice.bOperational THEN
	nErrorId := BACnet_ERR_OPERATIONAL;
	bReady := FALSE;

ELSIF _StatusFlags >= 4 THEN
	(* clear error flag *)
	nErrorId := BACnet_ERR_NO_ERROR;
	(* ready state *)
	bReady := TRUE;

	(* present value *)
	fPresentValue := _PresentValue;

	(* build bit states *)
	_StatusFlagsBits := F_BACnet_StatusFlags(_StatusFlags);

	(* copy states to output *)
	bOverridden := _StatusFlagsBits.overridden;
	bOutOfService := _StatusFlagsBits.out_of_service;
	bFault := _StatusFlagsBits.fault;
	bInAlarm := _StatusFlagsBits.in_alarm;
ELSE
	(* server device not ready, reset local ready also *)
	bReady := FALSE;
	(* and set error ID *)
	nErrorId := BACnet_ERR_WRONG_MAPPING;
END_IF

(* set error flag *)
bError := (nErrorId <> BACnet_ERR_NO_ERROR);

END_FUNCTION_BLOCK

// POUs/BACnet Objects/Remote (Client)/FB_BACnet_RemoteAnalogOutput
FUNCTION_BLOCK FB_BACnet_RemoteAnalogOutput
VAR_IN_OUT
	RemoteDevice		: FB_BACnet_RemoteDevice;
END_VAR
VAR_OUTPUT
	bReady				: BOOL;
	fPresentValue		: REAL;
	bOverridden			: BOOL;
	bOutOfService		: BOOL;
	bFault				: BOOL;
	bInAlarm			: BOOL;
	bError				: BOOL;
	nErrorId			: UINT;
END_VAR
VAR
	_PresentValue AT%I*: REAL; 			(* ~(BACnet_PresentValue 				:		: )
								   			(BACnet_ObjectType 					: AO	: )
											(BACnet_RemoteCycletimeRead 		: 1000	: )
											(BACnet_RemoteFlagsRead        		: 1		: )
											(BACnet_RemoteResubscriptionInterval: 240	: )
	                                		(BACnet_RemoteCycleTimeWrite   		: 1000	: )
	                                		(BACnet_RemoteFlagsWrite       		: 1		: )	*)
	_StatusFlags AT%I*: WORD; 			(* ~(BACnet_StatusFlags 				:		: )	*)
	_StatusFlagsBits : ST_BACnet_StatusFlags;

	_nUpdateCount : UDINT := 0;
END_VAR

(* update client device *)
IF RemoteDevice._nUpdateCount = _nUpdateCount THEN
	RemoteDevice();
END_IF
(* remind current number of update counter *)
_nUpdateCount := RemoteDevice._nUpdateCount;

IF RemoteDevice.bFirstCycle THEN
	(* first call of the server device since reboot/reset *)
	bReady := FALSE;

ELSIF NOT RemoteDevice.bOperational THEN
	nErrorId := BACnet_ERR_OPERATIONAL;
	bReady := FALSE;

ELSIF _StatusFlags >= 4 THEN
	(* clear error flag *)
	nErrorId := BACnet_ERR_NO_ERROR;
	(* ready state *)
	bReady := TRUE;

	(* present value *)
	fPresentValue := _PresentValue;

	(* build bit states *)
	_StatusFlagsBits := F_BACnet_StatusFlags(_StatusFlags);

	(* copy states to output *)
	bOverridden := _StatusFlagsBits.overridden;
	bOutOfService := _StatusFlagsBits.out_of_service;
	bFault := _StatusFlagsBits.fault;
	bInAlarm := _StatusFlagsBits.in_alarm;
ELSE
	(* server device not ready, reset local ready also *)
	bReady := FALSE;
	(* and set error ID *)
	nErrorId := BACnet_ERR_WRONG_MAPPING;
END_IF

(* set error flag *)
bError := (nErrorId <> BACnet_ERR_NO_ERROR);

END_FUNCTION_BLOCK

// POUs/BACnet Objects/Remote (Client)/FB_BACnet_RemoteAnalogValue
FUNCTION_BLOCK FB_BACnet_RemoteAnalogValue
VAR_IN_OUT
	RemoteDevice		: FB_BACnet_RemoteDevice;
END_VAR
VAR_OUTPUT
	bReady				: BOOL;
	fPresentValue		: REAL;
	bOverridden			: BOOL;
	bOutOfService		: BOOL;
	bFault				: BOOL;
	bInAlarm			: BOOL;
	bError				: BOOL;
	nErrorId			: UINT;
END_VAR
VAR
	_PresentValue AT%I*: REAL; 			(* ~(BACnet_PresentValue 				:		: )
								   			(BACnet_ObjectType 					: AV	: )
											(BACnet_RemoteCycletimeRead 		: 1000	: )
											(BACnet_RemoteFlagsRead        		: 1		: )
											(BACnet_RemoteResubscriptionInterval: 240	: )
	                                		(BACnet_RemoteCycleTimeWrite   		: 1000	: )
	                                		(BACnet_RemoteFlagsWrite       		: 1		: )	*)
	_StatusFlags AT%I*: WORD; 			(* ~(BACnet_StatusFlags 				:		: )	*)
	_StatusFlagsBits : ST_BACnet_StatusFlags;

	_nUpdateCount : UDINT := 0;
END_VAR

(* update client device *)
IF RemoteDevice._nUpdateCount = _nUpdateCount THEN
	RemoteDevice();
END_IF
(* remind current number of update counter *)
_nUpdateCount := RemoteDevice._nUpdateCount;

IF RemoteDevice.bFirstCycle THEN
	(* first call of the server device since reboot/reset *)
	bReady := FALSE;

ELSIF NOT RemoteDevice.bOperational THEN
	nErrorId := BACnet_ERR_OPERATIONAL;
	bReady := FALSE;

ELSIF _StatusFlags >= 4 THEN
	(* clear error flag *)
	nErrorId := BACnet_ERR_NO_ERROR;
	(* ready state *)
	bReady := TRUE;

	(* present value *)
	fPresentValue := _PresentValue;

	(* build bit states *)
	_StatusFlagsBits := F_BACnet_StatusFlags(_StatusFlags);

	(* copy states to output *)
	bOverridden := _StatusFlagsBits.overridden;
	bOutOfService := _StatusFlagsBits.out_of_service;
	bFault := _StatusFlagsBits.fault;
	bInAlarm := _StatusFlagsBits.in_alarm;
ELSE
	(* server device not ready, reset local ready also *)
	bReady := FALSE;
	(* and set error ID *)
	nErrorId := BACnet_ERR_WRONG_MAPPING;
END_IF

(* set error flag *)
bError := (nErrorId <> BACnet_ERR_NO_ERROR);

END_FUNCTION_BLOCK

// POUs/BACnet Objects/Remote (Client)/FB_BACnet_RemoteAveraging
FUNCTION_BLOCK FB_BACnet_RemoteAveraging
VAR_IN_OUT
	RemoteDevice		: FB_BACnet_RemoteDevice;
END_VAR
VAR_OUTPUT
	bReady				: BOOL;
	nAverageValue		: REAL;
	bError				: BOOL;
	nErrorId			: UINT;
END_VAR
VAR
	_AverageValue AT%I*: REAL; 		(* ~(BACnet_AverageValue 				:		: )
										(BACnet_ObjectType					: AVG  	: )
										(BACnet_RemoteCycletimeRead 		: 1000	: )
										(BACnet_RemoteFlagsRead        		: 1		: )
										(BACnet_RemoteResubscriptionInterval: 240	: )
										(BACnet_RemoteCycleTimeWrite   		: 1000	: )
										(BACnet_RemoteFlagsWrite       		: 1		: )	*)

	_nUpdateCount : UDINT := 0;
END_VAR

(* update client device *)
IF RemoteDevice._nUpdateCount = _nUpdateCount THEN
	RemoteDevice();
END_IF
(* remind current number of update counter *)
_nUpdateCount := RemoteDevice._nUpdateCount;

IF RemoteDevice.bOperational THEN
	(* clear error flag *)
	nErrorId := BACnet_ERR_NO_ERROR;
	(* ready state *)
	bReady := TRUE;
	(* present value *)
	nAverageValue := _AverageValue;
ELSE
	(* server device not ready, reset local ready also *)
	bReady := FALSE;
	(* and set error ID *)
	nErrorId := BACnet_ERR_OPERATIONAL;
END_IF

(* set error flag *)
bError := (nErrorId <> BACnet_ERR_NO_ERROR);

END_FUNCTION_BLOCK

// POUs/BACnet Objects/Remote (Client)/FB_BACnet_RemoteBinaryInput
FUNCTION_BLOCK FB_BACnet_RemoteBinaryInput
VAR_OUTPUT
	bReady				: BOOL;
	bPresentValue		: BOOL;
	bOverridden			: BOOL;
	bOutOfService		: BOOL;
	bFault				: BOOL;
	bInAlarm			: BOOL;
	bError				: BOOL;
	nErrorId			: UINT;
END_VAR
VAR_IN_OUT
	RemoteDevice			: FB_BACnet_RemoteDevice;
END_VAR
VAR
	_PresentValue AT%I*: WORD; 				(* ~(BACnet_PresentValue 				:		: )
												(BACnet_ObjectType					: BI    : )
												(BACnet_RemoteCycletimeRead 		: 1000	: )
												(BACnet_RemoteFlagsRead        		: 1		: )
												(BACnet_RemoteResubscriptionInterval: 240	: )
		                                		(BACnet_RemoteCycleTimeWrite   		: 1000	: )
		                                		(BACnet_RemoteFlagsWrite       		: 1		: )	*)
	_StatusFlags AT%I*: WORD; 				(* ~(BACnet_StatusFlags 				:	    : )	*)
	_StatusFlagsBits : ST_BACnet_StatusFlags;
	_nUpdateCount : UDINT := 0;
END_VAR

(* update client device *)
IF RemoteDevice._nUpdateCount = _nUpdateCount THEN
	RemoteDevice();
END_IF
(* remind current number of update counter *)
_nUpdateCount := RemoteDevice._nUpdateCount;

IF NOT RemoteDevice.bOperational THEN
	nErrorId := BACnet_ERR_OPERATIONAL;
	bReady := FALSE;

ELSIF _StatusFlags >= 4 THEN
	(* clear error flag *)
	nErrorId := BACnet_ERR_NO_ERROR;
	(* ready state *)
	bReady := TRUE;

	(* present value *)
	bPresentValue := F_BinPV_To_Bool(TO_INT(_PresentValue));

	(* build bit states *)
	_StatusFlagsBits := F_BACnet_StatusFlags(_StatusFlags);

	(* copy states to output *)
	bOverridden := _StatusFlagsBits.overridden;
	bOutOfService := _StatusFlagsBits.out_of_service;
	bFault := _StatusFlagsBits.fault;
	bInAlarm := _StatusFlagsBits.in_alarm;

ELSE
	bReady := FALSE;
	(* and set error ID *)
	nErrorId := BACnet_ERR_WRONG_MAPPING;
END_IF

(* set error flag *)
bError := (nErrorId <> BACnet_ERR_NO_ERROR);

END_FUNCTION_BLOCK

// POUs/BACnet Objects/Remote (Client)/FB_BACnet_RemoteBinaryOutput
FUNCTION_BLOCK FB_BACnet_RemoteBinaryOutput
VAR_IN_OUT
	RemoteDevice		: FB_BACnet_RemoteDevice;
END_VAR
VAR_OUTPUT
	bReady				: BOOL;
	bPresentValue		: BOOL;
	bOverridden			: BOOL;
	bOutOfService		: BOOL;
	bFault				: BOOL;
	bInAlarm			: BOOL;
	bError				: BOOL;
	nErrorId			: UINT;
END_VAR
VAR
	_PresentValue AT%I*: WORD; 			(* ~(BACnet_PresentValue 				:		: )
								   			(BACnet_ObjectType 					: BO	: )
											(BACnet_RemoteCycletimeRead 		: 1000	: )
											(BACnet_RemoteFlagsRead        		: 1		: )
											(BACnet_RemoteResubscriptionInterval: 240	: )
		                            		(BACnet_RemoteCycleTimeWrite   		: 1000	: )
		                            		(BACnet_RemoteFlagsWrite       		: 1		: )	*)
	_StatusFlags AT%I*: WORD; 			(* ~(BACnet_StatusFlags 				:		: )	*)
	_StatusFlagsBits : ST_BACnet_StatusFlags;
	_nUpdateCount : UDINT := 0;
END_VAR

(* update client device *)
IF RemoteDevice._nUpdateCount = _nUpdateCount THEN
	RemoteDevice();
END_IF
(* remind current number of update counter *)
_nUpdateCount := RemoteDevice._nUpdateCount;

IF RemoteDevice.bFirstCycle THEN
	(* first call of the server device since reboot/reset *)
	bReady := FALSE;

ELSIF NOT RemoteDevice.bOperational THEN
	nErrorId := BACnet_ERR_OPERATIONAL;
	bReady := FALSE;

ELSIF _StatusFlags >= 4 THEN
	(* clear error flag *)
	nErrorId := BACnet_ERR_NO_ERROR;
	(* ready state *)
	bReady := TRUE;

	(* present value *)
	bPresentValue := F_BinPV_To_Bool(TO_INT(_PresentValue));

	(* build bit states *)
	_StatusFlagsBits := F_BACnet_StatusFlags(_StatusFlags);

	(* copy states to output *)
	bOverridden := _StatusFlagsBits.overridden;
	bOutOfService := _StatusFlagsBits.out_of_service;
	bFault := _StatusFlagsBits.fault;
	bInAlarm := _StatusFlagsBits.in_alarm;
ELSE
	(* server device not ready, reset local ready also *)
	bReady := FALSE;
	(* and set error ID *)
	nErrorId := BACnet_ERR_WRONG_MAPPING;
END_IF

(* set error flag *)
bError := (nErrorId <> BACnet_ERR_NO_ERROR);

END_FUNCTION_BLOCK

// POUs/BACnet Objects/Remote (Client)/FB_BACnet_RemoteBinaryValue
FUNCTION_BLOCK FB_BACnet_RemoteBinaryValue
VAR_IN_OUT
	RemoteDevice		: FB_BACnet_RemoteDevice;
END_VAR
VAR_OUTPUT
	bReady				: BOOL;
	bPresentValue		: BOOL;
	bOverridden			: BOOL;
	bOutOfService		: BOOL;
	bFault				: BOOL;
	bInAlarm			: BOOL;
	bError				: BOOL;
	nErrorId			: UINT;
END_VAR
VAR

	_PresentValue AT%I*: WORD; 			(* ~(BACnet_PresentValue 				:		: )
								   			(BACnet_ObjectType 					: BV	: )
											(BACnet_RemoteCycletimeRead 		: 1000	: )
											(BACnet_RemoteFlagsRead        		: 1		: )
											(BACnet_RemoteResubscriptionInterval: 240	: )
	                                		(BACnet_RemoteCycleTimeWrite   		: 1000	: )
	                                		(BACnet_RemoteFlagsWrite       		: 1		: )	*)
	_StatusFlags AT%I*: WORD; 			(* ~(BACnet_StatusFlags 				:		: )	*)
	_StatusFlagsBits : ST_BACnet_StatusFlags;

	_nUpdateCount : UDINT := 0;
END_VAR

(* update client device *)
IF RemoteDevice._nUpdateCount = _nUpdateCount THEN
	RemoteDevice();
END_IF
(* remind current number of update counter *)
_nUpdateCount := RemoteDevice._nUpdateCount;

IF RemoteDevice.bFirstCycle THEN
	(* first call of the server device since reboot/reset *)
	bReady := FALSE;

ELSIF NOT RemoteDevice.bOperational THEN
	nErrorId := BACnet_ERR_OPERATIONAL;
	bReady := FALSE;

ELSIF _StatusFlags >= 4 THEN
	(* clear error flag *)
	nErrorId := BACnet_ERR_NO_ERROR;
	(* ready state *)
	bReady := TRUE;

	(* present value *)
	bPresentValue := F_BinPV_To_Bool(TO_INT(_PresentValue));

	(* build bit states *)
	_StatusFlagsBits := F_BACnet_StatusFlags(_StatusFlags);

	(* copy states to output *)
	bOverridden := _StatusFlagsBits.overridden;
	bOutOfService := _StatusFlagsBits.out_of_service;
	bFault := _StatusFlagsBits.fault;
	bInAlarm := _StatusFlagsBits.in_alarm;

ELSE
	(* server device not ready, reset local ready also *)
	bReady := FALSE;
	(* and set error ID *)
	nErrorId := BACnet_ERR_WRONG_MAPPING;
END_IF

(* set error flag *)
bError := (nErrorId <> BACnet_ERR_NO_ERROR);

END_FUNCTION_BLOCK

// POUs/BACnet Objects/Remote (Client)/FB_BACnet_RemoteCalendar
FUNCTION_BLOCK FB_BACnet_RemoteCalendar
VAR_IN_OUT
	RemoteDevice		: FB_BACnet_RemoteDevice;
END_VAR
VAR_OUTPUT
	bReady				: BOOL;
	bPresentValue		: BOOL;
	bError				: BOOL;
	nErrorId			: UINT;
END_VAR
VAR
	_PresentValue AT%I*: BOOL;	(* ~(BACnet_PresentValue 				:		: )
									(BACnet_ObjectType 					: CAL	: )
									(BACnet_RemoteCycletimeRead 		: 1000	: )
									(BACnet_RemoteFlagsRead        		: 1		: )
									(BACnet_RemoteResubscriptionInterval: 240	: )
                            		(BACnet_RemoteCycleTimeWrite   		: 1000	: )
                            		(BACnet_RemoteFlagsWrite       		: 1		: )	*)
	_nUpdateCount : UDINT := 0;
END_VAR

(* update client device *)
IF RemoteDevice._nUpdateCount = _nUpdateCount THEN
	RemoteDevice();
END_IF
(* remind current number of update counter *)
_nUpdateCount := RemoteDevice._nUpdateCount;

IF RemoteDevice.bOperational THEN
	(* clear error flag *)
	nErrorId := BACnet_ERR_NO_ERROR;
	(* ready state *)
	bReady := TRUE;
	(* present value *)
	bPresentValue := _PresentValue;
ELSE
	(* server device not ready, reset local ready also *)
	bReady := FALSE;
	(* and set error ID *)
	nErrorId := BACnet_ERR_OPERATIONAL;
END_IF

(* set error flag *)
bError := (nErrorId <> BACnet_ERR_NO_ERROR);

END_FUNCTION_BLOCK

// POUs/BACnet Objects/Remote (Client)/FB_BACnet_RemoteCommand
FUNCTION_BLOCK FB_BACnet_RemoteCommand
VAR_IN_OUT
	RemoteDevice		: FB_BACnet_RemoteDevice;
END_VAR
VAR_OUTPUT
	bReady				: BOOL;
	nPresentValue		: UDINT;
	bAllWritesOk		: BOOL; (* all actions in selected action list are written *)
	bInProcess			: BOOL; (* object is busy *)
	bError				: BOOL;
	nErrorId			: UINT;
END_VAR
VAR
	_PresentValueIn AT%I*: UDINT; 		(* ~(BACnet_PresentValue 				:		: )
								   			(BACnet_ObjectType 					: CMD	: )
											(BACnet_RemoteCycletimeRead 		: 1000	: )
											(BACnet_RemoteFlagsRead        		: 1		: )
											(BACnet_RemoteResubscriptionInterval: 240	: )
	                                		(BACnet_RemoteCycleTimeWrite   		: 1000	: )
	                                		(BACnet_RemoteFlagsWrite       		: 1		: )	*)
	_InProcess AT%I*: BOOL;				(* ~(BACnet_InProcess 					:		: )	*)
	_AllWritesSuccessful AT%I*: BOOL;	(* ~(BACnet_AllWritesSuccessful			:		: )	*)
	_nUpdateCount : UDINT := 0;
	_rtrigRetriggerPv : R_TRIG;
END_VAR

(* update client device *)
IF RemoteDevice._nUpdateCount = _nUpdateCount THEN
	RemoteDevice();
END_IF
(* remind current number of update counter *)
_nUpdateCount := RemoteDevice._nUpdateCount;

IF RemoteDevice.bOperational THEN
	(* clear error flag *)
	nErrorId := BACnet_ERR_NO_ERROR;
	(* ready state *)
	bReady := TRUE;
	(* present value from BACnet *)
	nPresentValue := _PresentValueIn;

	(* other states *)
	bAllWritesOk := _AllWritesSuccessful;
	bInProcess := _InProcess;
ELSIF RemoteDevice.bFirstCycle THEN
	(* first call of the server device since reboot/reset *)
	bReady := FALSE;
ELSE
	(* server device not ready, reset local ready also *)
	bReady := FALSE;
	(* and set error ID *)
	nErrorId := BACnet_ERR_WRONG_MAPPING;
END_IF

(* set error flag *)
bError := (nErrorId <> BACnet_ERR_NO_ERROR);

END_FUNCTION_BLOCK

// POUs/BACnet Objects/Remote (Client)/FB_BACnet_RemoteEventEnrollment
FUNCTION_BLOCK FB_BACnet_RemoteEventEnrollment
VAR_IN_OUT
	RemoteDevice		: FB_BACnet_RemoteDevice;
END_VAR
VAR_OUTPUT
	bReady				: BOOL;
	bError				: BOOL;
	nErrorId			: UINT;
END_VAR
VAR
	_ObjectType: E_BACNETOBJECTTYPE;	(* ~ (BACNET_OBJECTTYPE : EE : )	*)
	_nUpdateCount : UDINT := 0;
END_VAR

_ObjectType := BACnetObjectType_EventEnrollment;
(* update client device *)
IF RemoteDevice._nUpdateCount = _nUpdateCount THEN
	RemoteDevice();
END_IF
(* remind current number of update counter *)
_nUpdateCount := RemoteDevice._nUpdateCount;

IF RemoteDevice.bOperational THEN
	(* clear error flag *)
	nErrorId := BACnet_ERR_NO_ERROR;
	(* ready state *)
	bReady := TRUE;
ELSE
	(* server device not ready, reset local ready also *)
	bReady := FALSE;
	(* and set error ID *)
	nErrorId := BACnet_ERR_OPERATIONAL;
END_IF

(* set error flag *)
bError := (nErrorId <> BACnet_ERR_NO_ERROR);

END_FUNCTION_BLOCK

// POUs/BACnet Objects/Remote (Client)/FB_BACnet_RemoteFile
FUNCTION_BLOCK FB_BACnet_RemoteFile
VAR_IN_OUT
	RemoteDevice		: FB_BACnet_RemoteDevice;
END_VAR
VAR_OUTPUT
	bReady				: BOOL;
	fFileSize			: UDINT;
	bError				: BOOL;
	nErrorId			: UINT;
END_VAR
VAR
	_FileSize 			AT%I*: UDINT; 	(* ~(BACnet_FileSize 					:		: )
					   						(BACnet_ObjectType 					: FILE	: )
											(BACnet_RemoteCycletimeRead 		: 1000	: )
											(BACnet_RemoteFlagsRead        		: 1		: )
											(BACnet_RemoteResubscriptionInterval: 240	: )
	                                		(BACnet_RemoteCycleTimeWrite   		: 1000	: )
	                                		(BACnet_RemoteFlagsWrite       		: 1		: )	*)
	_nUpdateCount		: UDINT := 0;
END_VAR

(* update client device *)
IF RemoteDevice._nUpdateCount = _nUpdateCount THEN
	RemoteDevice();
END_IF
(* remind current number of update counter *)
_nUpdateCount := RemoteDevice._nUpdateCount;

IF RemoteDevice.bOperational THEN
	(* clear error flag *)
	nErrorId := BACnet_ERR_NO_ERROR;
	(* ready state *)
	bReady := TRUE;
	fFileSize := _FileSize;
ELSE
	(* server device not ready, reset local ready also *)
	bReady := FALSE;
	(* and set error ID *)
	nErrorId := BACnet_ERR_OPERATIONAL;
END_IF

(* set error flag *)
bError := (nErrorId <> BACnet_ERR_NO_ERROR);

END_FUNCTION_BLOCK

// POUs/BACnet Objects/Remote (Client)/FB_BACnet_RemoteGroup
FUNCTION_BLOCK FB_BACnet_RemoteGroup
VAR_IN_OUT
	RemoteDevice		: FB_BACnet_RemoteDevice;
END_VAR
VAR_OUTPUT
	bReady				: BOOL;
	bError				: BOOL;
	nErrorId			: UINT;
END_VAR
VAR
	_ObjectType: E_BACNETOBJECTTYPE;	(* ~ (BACNET_OBJECTTYPE : GROUP : )	*)
	_nUpdateCount : UDINT := 0;
END_VAR

_ObjectType := BACnetObjectType_Group;
(* update client device *)
IF RemoteDevice._nUpdateCount = _nUpdateCount THEN
	RemoteDevice();
END_IF
(* remind current number of update counter *)
_nUpdateCount := RemoteDevice._nUpdateCount;

IF RemoteDevice.bOperational THEN
	(* clear error flag *)
	nErrorId := BACnet_ERR_NO_ERROR;
	(* ready state *)
	bReady := TRUE;
ELSE
	(* server device not ready, reset local ready also *)
	bReady := FALSE;
	(* and set error ID *)
	nErrorId := BACnet_ERR_OPERATIONAL;
END_IF

(* set error flag *)
bError := (nErrorId <> BACnet_ERR_NO_ERROR);

END_FUNCTION_BLOCK

// POUs/BACnet Objects/Remote (Client)/FB_BACnet_RemoteLoop
FUNCTION_BLOCK FB_BACnet_RemoteLoop
VAR_IN_OUT
	RemoteDevice		: FB_BACnet_RemoteDevice;
END_VAR
VAR_OUTPUT
	bReady				: BOOL;
	fControlledValue	: REAL;
	fPresentValue		: REAL;
	bOverridden			: BOOL;
	bOutOfService		: BOOL;
	bFault				: BOOL;
	bInAlarm			: BOOL;
	bError				: BOOL;
	nErrorId			: UINT;
END_VAR
VAR
	_PresentValue AT%I*: REAL; 				(* ~(BACnet_PresentValue 				: 		: )
												(BACnet_ObjectType					: LOOP	: )
			                                	(BACnet_RemoteCycletimeRead 		: 1000	: )
												(BACnet_RemoteFlagsRead        		: 1     : )
                                   				(BACnet_RemoteResubscriptionInterval: 240 	: )
		                                		(BACnet_RemoteCycleTimeWrite   		: 1000	: )
		                                		(BACnet_RemoteFlagsWrite       		: 1		: )	*)
	_ControlledVariableValue AT%I*: REAL; 	(* ~(BACnet_ControlledVariableValue 	:		: )	*)
	_StatusFlags AT%I*: WORD; 				(* ~(BACnet_StatusFlags 				:		: )	*)
	_StatusFlagsBits : ST_BACnet_StatusFlags;
	_nUpdateCount : UDINT := 0;
END_VAR

(* update client device *)
IF RemoteDevice._nUpdateCount = _nUpdateCount THEN
	RemoteDevice();
END_IF
(* remind current number of update counter *)
_nUpdateCount := RemoteDevice._nUpdateCount;

IF NOT RemoteDevice.bOperational THEN
	nErrorId := BACnet_ERR_OPERATIONAL;
	bReady := FALSE;

ELSIF _StatusFlags >= 4 THEN
	(* clear error flag *)
	nErrorId := BACnet_ERR_NO_ERROR;
	(* ready state *)
	bReady := TRUE;

	(* present value *)
	fPresentValue := _PresentValue;
	fControlledValue := _ControlledVariableValue;

	(* build bit states *)
	_StatusFlagsBits := F_BACnet_StatusFlags(_StatusFlags);

	(* copy states to output *)
	bOverridden := _StatusFlagsBits.overridden;
	bOutOfService := _StatusFlagsBits.out_of_service;
	bFault := _StatusFlagsBits.fault;
	bInAlarm := _StatusFlagsBits.in_alarm;
ELSE
	(* server device not ready, reset local ready also *)
	bReady := FALSE;
	(* and set error ID *)
	nErrorId := BACnet_ERR_WRONG_MAPPING;
END_IF

(* set error flag *)
bError := (nErrorId <> BACnet_ERR_NO_ERROR);

END_FUNCTION_BLOCK

// POUs/BACnet Objects/Remote (Client)/FB_BACnet_RemoteMultiStateInput
FUNCTION_BLOCK FB_BACnet_RemoteMultiStateInput
VAR_IN_OUT
	RemoteDevice		: FB_BACnet_RemoteDevice;
END_VAR
VAR_OUTPUT
	bReady				: BOOL;
	nPresentValue		: UDINT;
	bOverridden			: BOOL;
	bOutOfService		: BOOL;
	bFault				: BOOL;
	bInAlarm			: BOOL;
	bError				: BOOL;
	nErrorId			: UINT;
END_VAR
VAR
	_PresentValue AT%I*: UDINT; 	(* ~(BACnet_PresentValue 				:		: )
								   		(BACnet_ObjectType 					: MI	: )
										(BACnet_RemoteCycletimeRead 		: 1000	: )
										(BACnet_RemoteFlagsRead        		: 1		: )
										(BACnet_RemoteResubscriptionInterval: 240	: )
                                		(BACnet_RemoteCycleTimeWrite   		: 1000	: )
                                		(BACnet_RemoteFlagsWrite       		: 1		: )	*)
	_StatusFlags AT%I*: WORD; 		(* ~(BACnet_StatusFlags 				:		: )	*)
	_StatusFlagsBits : ST_BACnet_StatusFlags;
	_nUpdateCount : UDINT := 0;
END_VAR

(* update client device *)
IF RemoteDevice._nUpdateCount = _nUpdateCount THEN
	RemoteDevice();
END_IF
(* remind current number of update counter *)
_nUpdateCount := RemoteDevice._nUpdateCount;

IF NOT RemoteDevice.bOperational THEN
	nErrorId := BACnet_ERR_OPERATIONAL;
	bReady := FALSE;

ELSIF _StatusFlags >= 4 THEN
	(* clear error flag *)
	nErrorId := BACnet_ERR_NO_ERROR;
	(* ready state *)
	bReady := TRUE;

	(* present value *)
	nPresentValue := _PresentValue;

	(* build bit states *)
	_StatusFlagsBits := F_BACnet_StatusFlags(_StatusFlags);

	(* copy states to output *)
	bOverridden := _StatusFlagsBits.overridden;
	bOutOfService := _StatusFlagsBits.out_of_service;
	bFault := _StatusFlagsBits.fault;
	bInAlarm := _StatusFlagsBits.in_alarm;

ELSE
	(* server device not ready, reset local ready also *)
	bReady := FALSE;
	(* and set error ID *)
	nErrorId := BACnet_ERR_WRONG_MAPPING;
END_IF

(* set error flag *)
bError := (nErrorId <> BACnet_ERR_NO_ERROR);

END_FUNCTION_BLOCK

// POUs/BACnet Objects/Remote (Client)/FB_BACnet_RemoteMultiStateOutput
FUNCTION_BLOCK FB_BACnet_RemoteMultiStateOutput
VAR_IN_OUT
	RemoteDevice		: FB_BACnet_RemoteDevice;
END_VAR
VAR_OUTPUT
	bReady				: BOOL;
	nPresentValue		: UDINT;
	bOverridden			: BOOL;
	bOutOfService		: BOOL;
	bFault				: BOOL;
	bInAlarm			: BOOL;
	nNbrOfStates		: UDINT;
	bError				: BOOL;
	nErrorId			: UINT;
END_VAR
VAR
	_PresentValue AT%I*: UDINT; 			(* ~(BACnet_PresentValue 				:		: )
								   				(BACnet_ObjectType					: MO	: )
												(BACnet_RemoteCycletimeRead 		: 1000	: )
												(BACnet_RemoteFlagsRead        		: 1		: )
												(BACnet_RemoteResubscriptionInterval: 240	: )
		                                		(BACnet_RemoteCycleTimeWrite   		: 1000	: )
		                                		(BACnet_RemoteFlagsWrite       		: 1		: )	*)
	_NumberOfStates AT%I*: UDINT;			(* ~(BACnet_NumberOfStates				:		: )	*)
	_StatusFlags AT%I*: WORD; 				(* ~(BACnet_StatusFlags					:		: )	*)
	_StatusFlagsBits : ST_BACnet_StatusFlags;
	_nUpdateCount : UDINT := 0;
END_VAR

(* update client device *)
IF RemoteDevice._nUpdateCount = _nUpdateCount THEN
	RemoteDevice();
END_IF
(* remind current number of update counter *)
_nUpdateCount := RemoteDevice._nUpdateCount;

IF RemoteDevice.bFirstCycle THEN
	(* first call of the server device since reboot/reset *)
	bReady := FALSE;

ELSIF NOT RemoteDevice.bOperational THEN
	nErrorId := BACnet_ERR_OPERATIONAL;
	bReady := FALSE;

ELSIF _StatusFlags >= 4 THEN
	(* clear error flag *)
	nErrorId := BACnet_ERR_NO_ERROR;
	(* ready state *)
	bReady := TRUE;

	(* present value *)
	nPresentValue := _PresentValue;

	(* build bit states *)
	_StatusFlagsBits := F_BACnet_StatusFlags(_StatusFlags);

	(* copy states to output *)
	bOverridden := _StatusFlagsBits.overridden;
	bOutOfService := _StatusFlagsBits.out_of_service;
	bFault := _StatusFlagsBits.fault;
	bInAlarm := _StatusFlagsBits.in_alarm;

	(* number of states *)
	nNbrOfStates := _NumberOfStates;

ELSE
	(* server device not ready, reset local ready also *)
	bReady := FALSE;
	(* and set error ID *)
	nErrorId := BACnet_ERR_WRONG_MAPPING;
END_IF

(* set error flag *)
bError := (nErrorId <> BACnet_ERR_NO_ERROR);

END_FUNCTION_BLOCK

// POUs/BACnet Objects/Remote (Client)/FB_BACnet_RemoteMultiStateValue
FUNCTION_BLOCK FB_BACnet_RemoteMultiStateValue
VAR_IN_OUT
	RemoteDevice		: FB_BACnet_RemoteDevice;
END_VAR
VAR_OUTPUT
	bReady				: BOOL;
	nPresentValue		: UDINT;
	bOverridden			: BOOL;
	bOutOfService		: BOOL;
	bFault				: BOOL;
	bInAlarm			: BOOL;
	nNbrOfStates		: UDINT;
	bError				: BOOL;
	nErrorId			: UINT;
END_VAR
VAR
	_PresentValue AT%I*: UDINT; 			(* ~(BACnet_PresentValue 				:		: )
								   				(BACnet_ObjectType 					: MV	: )
												(BACnet_RemoteCycletimeRead 		: 1000	: )
												(BACnet_RemoteFlagsRead        		: 1		: )
												(BACnet_RemoteResubscriptionInterval: 240	: )
		                                		(BACnet_RemoteCycleTimeWrite   		: 1000	: )
		                                		(BACnet_RemoteFlagsWrite       		: 1		: )	*)
	_NumberOfStates AT%I*: UDINT;			(* ~(BACnet_NumberOfStates				:		: )	*)
	_StatusFlags AT%I*: WORD; 				(* ~(BACnet_StatusFlags 				:		: )	*)
	_StatusFlagsBits : ST_BACnet_StatusFlags;
	_nUpdateCount : UDINT := 0;
END_VAR

(* update client device *)
IF RemoteDevice._nUpdateCount = _nUpdateCount THEN
	RemoteDevice();
END_IF
(* remind current number of update counter *)
_nUpdateCount := RemoteDevice._nUpdateCount;

IF RemoteDevice.bFirstCycle THEN
	(* first call of the server device since reboot/reset *)
	bReady := FALSE;

ELSIF NOT RemoteDevice.bOperational THEN
	nErrorId := BACnet_ERR_OPERATIONAL;
	bReady := FALSE;

ELSIF _StatusFlags >= 4 THEN
	(* clear error flag *)
	nErrorId := BACnet_ERR_NO_ERROR;
	(* ready state *)
	bReady := TRUE;

	(* present value *)
	nPresentValue := _PresentValue;

	(* build bit states *)
	_StatusFlagsBits := F_BACnet_StatusFlags(_StatusFlags);

	(* copy states to output *)
	bOverridden := _StatusFlagsBits.overridden;
	bOutOfService := _StatusFlagsBits.out_of_service;
	bFault := _StatusFlagsBits.fault;
	bInAlarm := _StatusFlagsBits.in_alarm;

	(* number of states *)
	nNbrOfStates := _NumberOfStates;

ELSE
	(* server device not ready, reset local ready also *)
	bReady := FALSE;
	(* and set error ID *)
	nErrorId := BACnet_ERR_WRONG_MAPPING;
END_IF

(* set error flag *)
bError := (nErrorId <> BACnet_ERR_NO_ERROR);

END_FUNCTION_BLOCK

// POUs/BACnet Objects/Remote (Client)/FB_BACnet_RemoteNotificationClass
FUNCTION_BLOCK FB_BACnet_RemoteNotificationClass
VAR_IN_OUT
	RemoteDevice		: FB_BACnet_RemoteDevice;
END_VAR
VAR_OUTPUT
	bReady				: BOOL;
	bError				: BOOL;
	nErrorId			: UINT;
END_VAR
VAR
	_ObjectType : E_BACNETOBJECTTYPE; (* ~(BACNET_OBJECTTYPE :NC:)  *)
	_nUpdateCount : UDINT := 0;
END_VAR

_ObjectType := BACnetObjectType_NotificationClass;
(* update client device *)
IF RemoteDevice._nUpdateCount = _nUpdateCount THEN
	RemoteDevice();
END_IF
(* remind current number of update counter *)
_nUpdateCount := RemoteDevice._nUpdateCount;

IF RemoteDevice.bOperational THEN
	(* clear error flag *)
	nErrorId := BACnet_ERR_NO_ERROR;
	(* ready state *)
	bReady := TRUE;
ELSE
	(* server device not ready, reset local ready also *)
	bReady := FALSE;
	(* and set error ID *)
	nErrorId := BACnet_ERR_OPERATIONAL;
END_IF

(* set error flag *)
bError := (nErrorId <> BACnet_ERR_NO_ERROR);

END_FUNCTION_BLOCK

// POUs/BACnet Objects/Remote (Client)/FB_BACnet_RemoteProgram
FUNCTION_BLOCK FB_BACnet_RemoteProgram
VAR_IN_OUT
	RemoteDevice		: FB_BACnet_RemoteDevice;
END_VAR
VAR_OUTPUT
	bReady				: BOOL;
	ePrgState			: E_BACNETPROGRAMSTATE;
	ePrgReasonHalt		: E_BACNETPROGRAMERROR;
	bOverridden			: BOOL;
	bOutOfService		: BOOL;
	bFault				: BOOL;
	bInAlarm			: BOOL;
	bError				: BOOL;
	nErrorId			: UINT;
END_VAR
VAR
	_ProgramState AT%I*: WORD;			(* ~(BACnet_ProgramState 				:		: )
								   			(BACnet_ObjectType 					: PROG	: )
			                            	(BACnet_RemoteCycletimeRead 		: 1000	: )
											(BACnet_RemoteFlagsRead        		: 1    	: )
                                   			(BACnet_RemoteResubscriptionInterval: 240 	: )
	                                		(BACnet_RemoteCycleTimeWrite   		: 1000	: )
	                                		(BACnet_RemoteFlagsWrite       		: 1		: )	*)
	_ReasonForHalt AT%I*: WORD;			(* ~(BACnet_ReasonForHalt 				: 		: )	*)
	_StatusFlags AT%I*: WORD;			(* ~(BACnet_StatusFlags 				:		: )	*)
	_nUpdateCount : UDINT := 0;
	_StatusFlagsBits : ST_BACnet_StatusFlags;
END_VAR

(* update client device *)
IF RemoteDevice._nUpdateCount = _nUpdateCount THEN
	RemoteDevice();
END_IF
(* remind current number of update counter *)
_nUpdateCount := RemoteDevice._nUpdateCount;

IF RemoteDevice.bFirstCycle THEN
	(* first call of the server device since reboot/reset *)
	bReady := FALSE;

ELSIF NOT RemoteDevice.bOperational THEN
	nErrorId := BACnet_ERR_OPERATIONAL;
	bReady := FALSE;

ELSIF _StatusFlags >= 4 THEN
	(* clear error flag *)
	nErrorId := BACnet_ERR_NO_ERROR;

	(* ready state *)
	bReady := TRUE;

	(* decode status flags *)
	_StatusFlagsBits := F_BACnet_StatusFlags(_StatusFlags);

	(* copy states to output *)
	bOverridden := _StatusFlagsBits.overridden;
	bOutOfService := _StatusFlagsBits.out_of_service;
	bFault := _StatusFlagsBits.fault;
	bInAlarm := _StatusFlagsBits.in_alarm;

	(* present value from BACnet *)
	ePrgState := TO_INT(_ProgramState);

	(* other states *)
	ePrgReasonHalt := to_int(_ReasonForHalt);
ELSE
	(* server device not ready, reset local ready also *)
	bReady := FALSE;
	(* and set error ID *)
	nErrorId := BACnet_ERR_WRONG_MAPPING;
END_IF

(* set error flag *)
bError := (nErrorId <> BACnet_ERR_NO_ERROR);

END_FUNCTION_BLOCK

// POUs/BACnet Objects/Remote (Client)/FB_BACnet_RemotePulseConverter
FUNCTION_BLOCK FB_BACnet_RemotePulseConverter
VAR_IN_OUT
	RemoteDevice		: FB_BACnet_RemoteDevice;
END_VAR
VAR_OUTPUT
	bReady				: BOOL;
	bOverridden			: BOOL;
	bOutOfService		: BOOL;
	bFault				: BOOL;
	bInAlarm			: BOOL;
	bError				: BOOL;
	nErrorId			: UINT;
END_VAR
VAR
	_StatusFlags AT%I*: UINT;		(* ~(BACnet_StatusFlags 				:		: )
										(BACnet_ObjectType 					: PC	: )
										(BACnet_RemoteCycletimeRead 		: 1000	: )
										(BACnet_RemoteFlagsRead        		: 1		: )
										(BACnet_RemoteResubscriptionInterval: 240	: )
                                		(BACnet_RemoteCycleTimeWrite   		: 1000	: )
                                		(BACnet_RemoteFlagsWrite       		: 1		: )	*)
	_StatusFlagsBits : ST_BACnet_StatusFlags;
	_nUpdateCount : UDINT := 0;
END_VAR

(* update client device *)
IF RemoteDevice._nUpdateCount = _nUpdateCount THEN
	RemoteDevice();
END_IF
(* remind current number of update counter *)
_nUpdateCount := RemoteDevice._nUpdateCount;

IF NOT RemoteDevice.bOperational THEN
	nErrorId := BACnet_ERR_OPERATIONAL;
	bReady := FALSE;

ELSIF _StatusFlags >= 4 THEN
	(* clear error flag *)
	nErrorId := BACnet_ERR_NO_ERROR;
	(* ready state *)
	bReady := TRUE;

	(* build bit states *)
	_StatusFlagsBits := F_BACnet_StatusFlags(_StatusFlags);

	(* copy states to output *)
	bOverridden := _StatusFlagsBits.overridden;
	bOutOfService := _StatusFlagsBits.out_of_service;
	bFault := _StatusFlagsBits.fault;
	bInAlarm := _StatusFlagsBits.in_alarm;

ELSE
	(* server device not ready, reset local ready also *)
	bReady := FALSE;
	(* and set error ID *)
	nErrorId := BACnet_ERR_WRONG_MAPPING;
END_IF

(* set error flag *)
bError := (nErrorId <> BACnet_ERR_NO_ERROR);

END_FUNCTION_BLOCK

// POUs/BACnet Objects/Remote (Client)/FB_BACnet_RemoteSchedule
FUNCTION_BLOCK FB_BACnet_RemoteSchedule
VAR_IN_OUT
	RemoteDevice			: FB_BACnet_RemoteDevice;
END_VAR
VAR_OUTPUT
	bReady				: BOOL;
	bPresentValue		: BOOL;
	bOverridden			: BOOL;
	bOutOfService		: BOOL;
	bFault				: BOOL;
	bInAlarm			: BOOL;
	bError				: BOOL;
	nErrorId			: UINT;
END_VAR
VAR
	_StatusFlags AT%I*: WORD; 	(* ~(BACnet_StatusFlags 				:		: )	*)
	_PresentValue AT%I*: BOOL;	(* ~(BACnet_PresentValueBool 			:		: )
									(BACnet_ObjectType 					: SCHED	: )
									(BACnet_RemoteCycletimeRead 		: 1000	: )
									(BACnet_RemoteFlagsRead        		: 1		: )
									(BACnet_RemoteResubscriptionInterval: 240	: )
                            		(BACnet_RemoteCycleTimeWrite   		: 1000	: )
                            		(BACnet_RemoteFlagsWrite       		: 1		: )	*)
	_StatusFlagsBits : ST_BACnet_StatusFlags;
	_nUpdateCount : UDINT := 0;
END_VAR

(* update client device *)
IF RemoteDevice._nUpdateCount = _nUpdateCount THEN
	RemoteDevice();
END_IF
(* remind current number of update counter *)
_nUpdateCount := RemoteDevice._nUpdateCount;

IF NOT RemoteDevice.bOperational THEN
	nErrorId := BACnet_ERR_OPERATIONAL;
	bReady := FALSE;

ELSIF _StatusFlags >= 4 THEN
	(* clear error flag *)
	nErrorId := BACnet_ERR_NO_ERROR;
	(* ready state *)
	bReady := TRUE;

	(* present value *)
	bPresentValue := _PresentValue;

	(* build bit states *)
	_StatusFlagsBits := F_BACnet_StatusFlags(_StatusFlags);

	(* copy states to output *)
	bOverridden := _StatusFlagsBits.overridden;
	bOutOfService := _StatusFlagsBits.out_of_service;
	bFault := _StatusFlagsBits.fault;
	bInAlarm := _StatusFlagsBits.in_alarm;

ELSE
	bReady := FALSE;
	(* and set error ID *)
	nErrorId := BACnet_ERR_WRONG_MAPPING;
END_IF

(* set error flag *)
bError := (nErrorId <> BACnet_ERR_NO_ERROR);

END_FUNCTION_BLOCK

// POUs/BACnet Objects/Remote (Client)/FB_BACnet_RemoteTrendLog
FUNCTION_BLOCK FB_BACnet_RemoteTrendLog
VAR_IN_OUT
	RemoteDevice			: FB_BACnet_RemoteDevice;
END_VAR
VAR_OUTPUT
	bReady				: BOOL;
	bLogEnable			: BOOL;
	nRecordCount		: UDINT;
	nTotalCount			: UDINT;
	bError				: BOOL;
	nErrorId			: UINT;
END_VAR
VAR
	_RecordCount AT%I*: UDINT;		(* ~(BACnet_RecordCount					:		: )
										(BACnet_ObjectType					: TLOG	: )
										(BACnet_RemoteCycletimeRead 		: 1000	: )
										(BACnet_RemoteFlagsRead        		: 1		: )
										(BACnet_RemoteResubscriptionInterval: 240	: )
                                		(BACnet_RemoteCycleTimeWrite   		: 1000	: )
                                		(BACnet_RemoteFlagsWrite       		: 1		: )	*)
	_TotalRecordCount AT%I*: UDINT;	(* ~(BACnet_TotalRecordCount			:		: )	*)
	_LogEnable AT%I*: BOOL;			(* ~(BACnet_LogEnable					: 		: )	*)
	_nUpdateCount : UDINT := 0;
END_VAR

(* update client device *)
IF RemoteDevice._nUpdateCount = _nUpdateCount THEN
	RemoteDevice();
END_IF
(* remind current number of update counter *)
_nUpdateCount := RemoteDevice._nUpdateCount;

IF RemoteDevice.bOperational THEN
	(* clear error flag *)
	nErrorId := BACnet_ERR_NO_ERROR;
	(* ready state *)
	bReady := TRUE;

	(* other states *)
	nRecordCount := _RecordCount;
	nTotalCount := _TotalRecordCount;
	bLogEnable := _LogEnable;

ELSE
	bReady := FALSE;
	(* and set error ID *)
	nErrorId := BACnet_ERR_OPERATIONAL;
END_IF

(* set error flag *)
bError := (nErrorId <> BACnet_ERR_NO_ERROR);

END_FUNCTION_BLOCK

// POUs/BACnet Signals/FB_BACnet_PWM
FUNCTION_BLOCK FB_BACnet_PWM
VAR_INPUT
	bEnable			: BOOL;
	fPercent		: REAL; (* 0...100% *)
	tPeriod			: TIME; (* PWM period time *)
END_VAR
VAR_OUTPUT
	bEnablePV		: BOOL;
	bPresentValue	: BOOL;
END_VAR
VAR
	_fOut			: REAL;
	_tOn			: TIME;
	_tonPeriod		: TON;
	_tofOn			: TOF;
END_VAR

(* check limits *)
_fOut := LIMIT(0.0, fPercent, 100.0);

(* convert from percent value to time value in relation to period time (100% = tPara_Period, 0% = 0s) *)
_tOn := REAL_TO_TIME((_fOut / 100.0) * TIME_TO_REAL(tPeriod));

(* call period timer *)
_tonPeriod(
	IN	:= TRUE,
	PT	:= tPeriod,
	Q	=> ,
	ET	=> );

(* call on timer *)
_tofOn(
	IN	:= _tonPeriod.Q AND (_tOn > T#0ms),
	PT	:= _tOn,
	Q	=> ,
	ET	=> );

IF _tonPeriod.Q THEN
	_tonPeriod(IN:= FALSE);
	_tonPeriod(IN:= TRUE);
END_IF

(* set output *)
bPresentValue := (_tofOn.Q OR _tofOn.IN) AND bEnable;
bEnablePV := bEnable;

END_FUNCTION_BLOCK

// POUs/FB_BACnet_NotificationSink
FUNCTION_BLOCK FB_BACnet_NotificationSink
VAR_INPUT
	bReload			: BOOL;
	nAmsPort		: T_AmsPort := 0;
END_VAR
VAR_OUTPUT
	bReady			: BOOL;
	stBACnetAds		: ST_BACnet_AdsConnection;
END_VAR
VAR
	_rtrigReload	: R_TRIG;
	_nUpdateCountAdp: UDINT := 0;
	_BACnetAdapter	: POINTER TO FB_BACnet_Adapter;
END_VAR

(* check pointer to bacnet adapter instance *)
IF pBACnet_Adapter > 0 THEN
	_BACnetAdapter := pBACnet_Adapter;
ELSE
	_BACnetAdapter := ADR(fbBACnet_Adapter);
END_IF

(* update adapter *)
IF _BACnetAdapter^._nUpdateCount = _nUpdateCountAdp THEN
	_BACnetAdapter^();
END_IF
(* remind current number of update counter *)
_nUpdateCountAdp := _BACnetAdapter^._nUpdateCount;

(* set ads info *)
stBACnetAds.nAmsPort := nAmsPort;
stBACnetAds.bNSink := TRUE;
stBACnetAds.bServer := FALSE;
stBACnetAds.bClient := FALSE;
stBACnetAds.nDeviceId := 16#FFFFFFFF;
stBACnetAds.sAmsNetId := _BACnetAdapter^.sAmsNetId;
bReady := stBACnetAds.bValid;
stBACnetAds.bValid :=	(nAmsPort >= 1000) AND (nAmsPort < 16#FFFF)
					AND	(_BACnetAdapter^.eAdapterStatus > BACnetAdapterStatus_Init);

(* set reload counter *)
_rtrigReload(CLK:= bReload, Q=> );
IF stBACnetAds.bValid AND (_rtrigReload.Q OR (NOT bReady)) THEN
	stBACnetAds.nReload := stBACnetAds.nReload + 1;
END_IF

(* set states *)
bReady := stBACnetAds.bValid;

END_FUNCTION_BLOCK
